KUKA KRL program: MyProgram_147().src

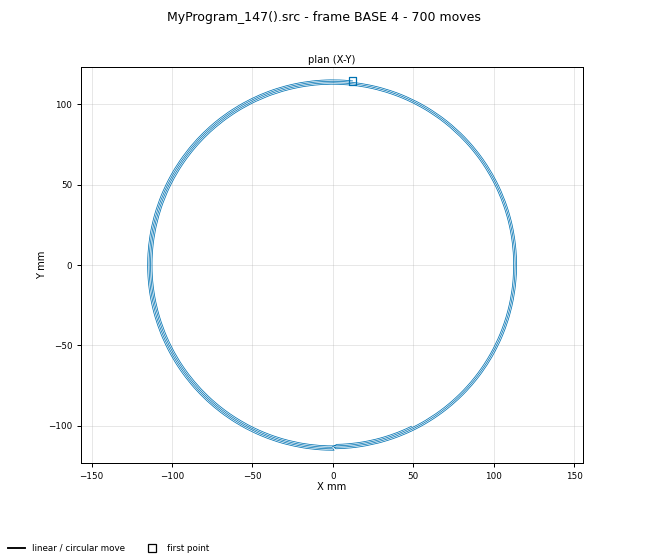
[picture p0: tool path of MyProgram_147().src in frame BASE 4, 700 of 700 moves have a stored position in this frame; points joined in program order, loops and branches not executed]
&ACCESS RVP
&REL 1
&PARAM TEMPLATE = C:\KRC\Roboter\Template\vorgabe
&PARAM EDITMASK = *
DEF MyProgram_147()
; ---- Setting reference (Base) ----
$BASE = BASE_DATA[4]

; --------------------------
; ---- Setting tool (TCP) ----
$TOOL = TOOL_DATA[3]
; --------------------------

$VEL.CP = VEL_APROX_PRINT
Startdeposition()
$VEL.CP = VEL_PRINT
LIN {X 12.2329,Y 114.5089,Z 116,A 79.5823,B 24.9341,C -1.8753,E1 25.0169,E2 366.2981} C_DIS
LIN {X 9.8806,Y 114.7378,Z 116,A 80.9993,B 24.9333,C -1.8859,E1 25.0129,E2 364.8568} C_DIS
LIN {X 7.0618,Y 114.9457,Z 116,A 82.4053,B 24.9333,C -1.8859,E1 25.0089,E2 363.4514} C_DIS
LIN {X 4.2388,Y 115.0844,Z 116,A 83.812,B 24.9333,C -1.8859,E1 25.005,E2 362.0453} C_DIS
LIN {X 1.3378,Y 115.1542,Z 116,A 85.1896,B 24.9335,C -1.8828,E1 25.0012,E2 360.6752} C_DIS
LIN {X -1.4132,Y 115.1537,Z 116,A 86.6253,B 24.9334,C -1.8854,E1 24.9972,E2 359.2332} C_DIS
LIN {X -4.2388,Y 115.0844,Z 116,A 88.0326,B 24.9334,C -1.885,E1 24.9932,E2 357.8267} C_DIS
LIN {X -7.0618,Y 114.9457,Z 116,A 89.4367,B 24.9334,C -1.8844,E1 24.9893,E2 356.4236} C_DIS
LIN {X -9.9557,Y 114.7308,Z 116,A 90.8528,B 24.9336,C -1.8826,E1 24.9854,E2 355.0113} C_DIS
LIN {X -12.7684,Y 114.452,Z 116,A 92.2606,B 24.9336,C -1.8819,E1 24.9815,E2 353.6042} C_DIS
LIN {X -15.5836,Y 114.1027,Z 116,A 93.7775,B 24.9334,C -1.8856,E1 24.9773,E2 352.0775} C_DIS
LIN {X -18.2945,Y 113.7,Z 116,A 95.072,B 24.9336,C -1.8816,E1 24.9737,E2 350.7912} C_DIS
LIN {X -21.0793,Y 113.2168,Z 116,A 96.4806,B 24.9336,C -1.8807,E1 24.9698,E2 349.3834} C_DIS
LIN {X -23.8514,Y 112.6654,Z 116,A 97.8569,B 24.9339,C -1.8782,E1 24.9661,E2 348.0114} C_DIS
LIN {X -26.6092,Y 112.0461,Z 116,A 99.2985,B 24.9339,C -1.8784,E1 24.9622,E2 346.5674} C_DIS
LIN {X -29.4238,Y 111.3397,Z 116,A 100.7129,B 24.934,C -1.8757,E1 24.9583,E2 345.1574} C_DIS
LIN {X -32.6132,Y 110.4458,Z 116,A 102.1625,B 24.9348,C -1.8656,E1 24.9545,E2 343.7295} C_DIS
LIN {X -34.8515,Y 109.7618,Z 116,A 103.4978,B 24.9343,C -1.8714,E1 24.9509,E2 342.378} C_DIS
LIN {X -37.5347,Y 108.8734,Z 116,A 104.9418,B 24.9343,C -1.8713,E1 24.9471,E2 340.9315} C_DIS
LIN {X -40.1953,Y 107.9195,Z 116,A 106.3522,B 24.9345,C -1.8696,E1 24.9434,E2 339.5222} C_DIS
LIN {X -42.8317,Y 106.9006,Z 116,A 107.7627,B 24.9345,C -1.8679,E1 24.9397,E2 338.1129} C_DIS
LIN {X -45.3731,Y 105.8474,Z 116,A 109.1681,B 24.9346,C -1.8674,E1 24.9361,E2 336.7052} C_DIS
LIN {X -48.0254,Y 104.6701,Z 116,A 110.5497,B 24.935,C -1.8627,E1 24.9326,E2 335.3316} C_DIS
LIN {X -50.5121,Y 103.4935,Z 116,A 111.9577,B 24.935,C -1.8621,E1 24.9291,E2 333.9213} C_DIS
LIN {X -53.1035,Y 102.1876,Z 116,A 113.4063,B 24.9352,C -1.86,E1 24.9255,E2 332.4739} C_DIS
LIN {X -55.5294,Y 100.8903,Z 116,A 114.7802,B 24.9353,C -1.8578,E1 24.9221,E2 331.1013} C_DIS
LIN {X -58.2622,Y 99.3355,Z 116,A 116.2478,B 24.9358,C -1.851,E1 24.9186,E2 329.6454} C_DIS
LIN {X -60.8906,Y 97.7458,Z 116,A 117.682,B 24.9362,C -1.8443,E1 24.9152,E2 328.2229} C_DIS
LIN {X -62.8639,Y 96.4905,Z 116,A 119.0192,B 24.9359,C -1.8492,E1 24.912,E2 326.8696} C_DIS
LIN {X -65.151,Y 94.9617,Z 116,A 120.4282,B 24.9359,C -1.8481,E1 24.9087,E2 325.4585} C_DIS
LIN {X -67.5228,Y 93.2896,Z 116,A 121.8441,B 24.9363,C -1.844,E1 24.9055,E2 324.0474} C_DIS
LIN {X -69.7321,Y 91.6505,Z 116,A 123.2858,B 24.9363,C -1.8442,E1 24.9023,E2 322.6003} C_DIS
LIN {X -71.9603,Y 89.9116,Z 116,A 124.6663,B 24.9365,C -1.84,E1 24.8993,E2 321.2244} C_DIS
LIN {X -74.1452,Y 88.1185,Z 116,A 126.0793,B 24.9367,C -1.8372,E1 24.8963,E2 319.8128} C_DIS
LIN {X -76.2854,Y 86.2724,Z 116,A 127.5247,B 24.9368,C -1.8356,E1 24.8932,E2 318.3655} C_DIS
LIN {X -78.4346,Y 84.3226,Z 116,A 128.9092,B 24.9372,C -1.8298,E1 24.8904,E2 316.9893} C_DIS
LIN {X -80.4267,Y 82.4253,Z 116,A 130.3516,B 24.9372,C -1.8295,E1 24.8875,E2 315.5414} C_DIS
LIN {X -82.4776,Y 80.3724,Z 116,A 131.7363,B 24.9377,C -1.8236,E1 24.8848,E2 314.165} C_DIS
LIN {X -84.3742,Y 78.3797,Z 116,A 133.1469,B 24.9377,C -1.8218,E1 24.8821,E2 312.7524} C_DIS
LIN {X -86.322,Y 76.2286,Z 116,A 134.5984,B 24.938,C -1.8185,E1 24.8794,E2 311.3024} C_DIS
LIN {X -88.1185,Y 74.1452,Z 116,A 135.975,B 24.9382,C -1.8152,E1 24.8769,E2 309.9273} C_DIS
LIN {X -89.9584,Y 71.9011,Z 116,A 137.427,B 24.9385,C -1.8118,E1 24.8743,E2 308.4768} C_DIS
LIN {X -91.6958,Y 69.6718,Z 116,A 138.8415,B 24.9387,C -1.8083,E1 24.8719,E2 307.0638} C_DIS
LIN {X -93.3342,Y 67.4619,Z 116,A 140.218,B 24.9389,C -1.8049,E1 24.8697,E2 305.6888} C_DIS
LIN {X -95.0009,Y 65.0932,Z 116,A 141.6704,B 24.9392,C -1.8013,E1 24.8674,E2 304.2377} C_DIS
LIN {X -96.5727,Y 62.7375,Z 116,A 143.0854,B 24.9394,C -1.7976,E1 24.8652,E2 302.8245} C_DIS
LIN {X -98.0441,Y 60.413,Z 116,A 144.4953,B 24.9396,C -1.7953,E1 24.8631,E2 301.4127} C_DIS
LIN {X -99.4972,Y 57.9887,Z 116,A 145.8778,B 24.9399,C -1.7903,E1 24.8611,E2 300.0351} C_DIS
LIN {X -100.8903,Y 55.5294,Z 116,A 147.4168,B 24.9399,C -1.7916,E1 24.859,E2 298.4851} C_DIS
LIN {X -102.257,Y 52.9696,Z 116,A 148.7117,B 24.9405,C -1.7813,E1 24.8574,E2 297.2078} C_DIS
LIN {X -103.5262,Y 50.4441,Z 116,A 150.1271,B 24.9408,C -1.7774,E1 24.8556,E2 295.794} C_DIS
LIN {X -104.733,Y 47.8883,Z 116,A 151.5769,B 24.941,C -1.7749,E1 24.8539,E2 294.3422} C_DIS
LIN {X -105.8474,Y 45.3731,Z 116,A 152.9548,B 24.9412,C -1.7711,E1 24.8524,E2 292.9658} C_DIS
LIN {X -106.929,Y 42.7618,Z 116,A 154.4259,B 24.9413,C -1.7694,E1 24.8508,E2 291.4906} C_DIS
LIN {X -107.9462,Y 40.1247,Z 116,A 155.8183,B 24.9417,C -1.7644,E1 24.8495,E2 290.1021} C_DIS
LIN {X -108.9055,Y 37.4426,Z 116,A 157.236,B 24.9419,C -1.76,E1 24.8482,E2 288.6869} C_DIS
LIN {X -109.785,Y 34.7797,Z 116,A 158.6502,B 24.9422,C -1.7564,E1 24.847,E2 287.2732} C_DIS
LIN {X -110.6055,Y 32.075,Z 116,A 160.066,B 24.9425,C -1.7523,E1 24.8458,E2 285.859} C_DIS
LIN {X -111.3781,Y 29.2779,Z 116,A 161.487,B 24.9428,C -1.7468,E1 24.8448,E2 284.4428} C_DIS
LIN {X -112.1254,Y 26.2662,Z 116,A 162.9247,B 24.9434,C -1.7376,E1 24.8439,E2 283.0187} C_DIS
LIN {X -112.6654,Y 23.8514,Z 116,A 164.3141,B 24.9433,C -1.74,E1 24.843,E2 281.6154} C_DIS
LIN {X -113.2168,Y 21.0793,Z 116,A 165.7301,B 24.9435,C -1.7358,E1 24.8423,E2 280.2009} C_DIS
LIN {X -113.7,Y 18.2945,Z 116,A 167.1465,B 24.9438,C -1.7317,E1 24.8417,E2 278.786} C_DIS
LIN {X -114.1812,Y 14.9855,Z 116,A 168.604,B 24.9447,C -1.718,E1 24.8411,E2 277.3523} C_DIS
LIN {X -114.4686,Y 12.6184,Z 116,A 169.9837,B 24.9444,C -1.7219,E1 24.8406,E2 275.9551} C_DIS
LIN {X -114.7378,Y 9.8806,Z 116,A 171.3948,B 24.9446,C -1.7192,E1 24.8403,E2 274.5421} C_DIS
LIN {X -114.9457,Y 7.0618,Z 116,A 172.8108,B 24.9449,C -1.715,E1 24.84,E2 273.1276} C_DIS
LIN {X -115.0844,Y 4.2388,Z 116,A 174.2271,B 24.9451,C -1.7108,E1 24.8399,E2 271.7126} C_DIS
LIN {X -115.1548,Y 1.2669,Z 116,A 175.6689,B 24.9456,C -1.7045,E1 24.8398,E2 270.2772} C_DIS
LIN {X -115.1537,Y -1.4132,Z 116,A 177.0592,B 24.9456,C -1.7025,E1 24.8398,E2 268.8834} C_DIS
LIN {X -115.0844,Y -4.2388,Z 116,A 178.6075,B 24.9456,C -1.7037,E1 24.84,E2 267.3229} C_DIS
LIN {X -114.9457,Y -7.0618,Z 116,A 179.8914,B 24.9462,C -1.6942,E1 24.8402,E2 266.054} C_DIS
LIN {X -114.7378,Y -9.8806,Z 116,A -178.7251,B 24.9466,C -1.6887,E1 24.8405,E2 264.6751} C_DIS
LIN {X -114.4607,Y -12.6935,Z 116,A -177.2766,B 24.9467,C -1.6859,E1 24.8409,E2 263.2246} C_DIS
LIN {X -114.1147,Y -15.4986,Z 116,A -175.8606,B 24.947,C -1.6818,E1 24.8414,E2 261.8099} C_DIS
LIN {X -113.7,Y -18.2945,Z 116,A -174.3898,B 24.9471,C -1.68,E1 24.842,E2 260.3348} C_DIS
LIN {X -113.2168,Y -21.0793,Z 116,A -173.0286,B 24.9475,C -1.6737,E1 24.8427,E2 258.9805} C_DIS
LIN {X -112.6654,Y -23.8514,Z 116,A -171.6455,B 24.9478,C -1.6684,E1 24.8435,E2 257.602} C_DIS
LIN {X -112.0461,Y -26.6092,Z 116,A -170.1971,B 24.948,C -1.6657,E1 24.8444,E2 256.1515} C_DIS
LIN {X -111.3397,Y -29.4238,Z 116,A -168.7763,B 24.9483,C -1.6603,E1 24.8454,E2 254.7352} C_DIS
LIN {X -110.584,Y -32.1473,Z 116,A -167.3609,B 24.9486,C -1.6564,E1 24.8465,E2 253.3209} C_DIS
LIN {X -109.7618,Y -34.8515,Z 116,A -165.9798,B 24.9489,C -1.6511,E1 24.8476,E2 251.9445} C_DIS
LIN {X -108.8984,Y -37.4635,Z 116,A -164.5353,B 24.9489,C -1.6501,E1 24.8489,E2 250.4943} C_DIS
LIN {X -107.8663,Y -40.3358,Z 116,A -163.142,B 24.9496,C -1.6405,E1 24.8502,E2 249.116} C_DIS
LIN {X -106.929,Y -42.7618,Z 116,A -161.6443,B 24.9493,C -1.6449,E1 24.8518,E2 247.5992} C_DIS
LIN {X -105.8474,Y -45.3731,Z 116,A -160.2896,B 24.9497,C -1.6387,E1 24.8533,E2 246.2517} C_DIS
LIN {X -104.6701,Y -48.0254,Z 116,A -158.9038,B 24.9501,C -1.6322,E1 24.8548,E2 244.8739} C_DIS
LIN {X -103.4935,Y -50.5121,Z 116,A -157.4923,B 24.9502,C -1.6301,E1 24.8566,E2 243.4598} C_DIS
LIN {X -102.2227,Y -53.0367,Z 116,A -156.0453,B 24.9503,C -1.6279,E1 24.8584,E2 242.0104} C_DIS
LIN {X -100.8903,Y -55.5294,Z 116,A -154.663,B 24.9506,C -1.623,E1 24.8602,E2 240.6324} C_DIS
LIN {X -99.2144,Y -58.4671,Z 116,A -153.1707,B 24.9514,C -1.6107,E1 24.8623,E2 239.1617} C_DIS
LIN {X -98.0441,Y -60.413,Z 116,A -151.8018,B 24.951,C -1.6175,E1 24.8643,E2 237.7696} C_DIS
LIN {X -96.4905,Y -62.8639,Z 116,A -150.4166,B 24.9514,C -1.6113,E1 24.8664,E2 236.3922} C_DIS
LIN {X -94.9186,Y -65.213,Z 116,A -149.0024,B 24.9516,C -1.608,E1 24.8686,E2 234.9787} C_DIS
LIN {X -93.2896,Y -67.5228,Z 116,A -147.5543,B 24.9516,C -1.6062,E1 24.871,E2 233.5278} C_DIS
LIN {X -91.6045,Y -69.7919,Z 116,A -146.1748,B 24.9519,C -1.6016,E1 24.8733,E2 232.1526} C_DIS
LIN {X -89.6717,Y -72.2564,Z 116,A -144.7035,B 24.9524,C -1.5943,E1 24.8758,E2 230.6918} C_DIS
LIN {X -88.0413,Y -74.2358,Z 116,A -143.3457,B 24.9524,C -1.5947,E1 24.8782,E2 229.3268} C_DIS
LIN {X -86.2724,Y -76.2854,Z 116,A -141.9056,B 24.9524,C -1.5954,E1 24.8809,E2 227.8785} C_DIS
LIN {X -84.3226,Y -78.4346,Z 116,A -140.5216,B 24.9526,C -1.5897,E1 24.8835,E2 226.502} C_DIS
LIN {X -82.4253,Y -80.4267,Z 116,A -139.0797,B 24.9526,C -1.5897,E1 24.8863,E2 225.0537} C_DIS
LIN {X -80.3724,Y -82.4776,Z 116,A -137.6961,B 24.953,C -1.5842,E1 24.889,E2 223.6776} C_DIS
LIN {X -78.3797,Y -84.3742,Z 116,A -136.1188,B 24.9526,C -1.5901,E1 24.8923,E2 222.0797} C_DIS
LIN {X -76.1041,Y -86.4307,Z 116,A -134.8247,B 24.9534,C -1.5774,E1 24.8949,E2 220.8108} C_DIS
LIN {X -74.1452,Y -88.1185,Z 116,A -133.4626,B 24.9534,C -1.578,E1 24.8979,E2 219.4418} C_DIS
LIN {X -71.9011,Y -89.9584,Z 116,A -131.8975,B 24.9532,C -1.5805,E1 24.9013,E2 217.8651} C_DIS
LIN {X -69.7321,Y -91.6505,Z 116,A -130.4675,B 24.9532,C -1.5805,E1 24.9045,E2 216.4296} C_DIS
LIN {X -67.4005,Y -93.378,Z 116,A -129.2239,B 24.9538,C -1.5696,E1 24.9072,E2 215.2078} C_DIS
LIN {X -65.0886,Y -95.004,Z 116,A -127.6193,B 24.9535,C -1.5757,E1 24.911,E2 213.5832} C_DIS
LIN {X -62.8009,Y -96.532,Z 116,A -126.3729,B 24.9539,C -1.5683,E1 24.9138,E2 212.3503} C_DIS
LIN {X -60.413,Y -98.0441,Z 116,A -124.994,B 24.9541,C -1.565,E1 24.9171,E2 210.975} C_DIS
LIN {X -57.9233,Y -99.5348,Z 116,A -123.4021,B 24.9539,C -1.5692,E1 24.921,E2 209.3683} C_DIS
LIN {X -55.5294,Y -100.8903,Z 116,A -122.1408,B 24.9542,C -1.5627,E1 24.924,E2 208.1187} C_DIS
LIN {X -52.9696,Y -102.257,Z 116,A -120.7254,B 24.9544,C -1.5596,E1 24.9275,E2 206.7067} C_DIS
LIN {X -50.4441,Y -103.5262,Z 116,A -119.3494,B 24.9546,C -1.5566,E1 24.9309,E2 205.3343} C_DIS
LIN {X -47.957,Y -104.702,Z 116,A -117.9108,B 24.9546,C -1.558,E1 24.9346,E2 203.8888} C_DIS
LIN {X -45.3036,Y -105.8767,Z 116,A -116.496,B 24.9546,C -1.5552,E1 24.9382,E2 202.4773} C_DIS
LIN {X -42.6916,Y -106.9566,Z 116,A -115.1207,B 24.9548,C -1.5524,E1 24.9418,E2 201.1055} C_DIS
LIN {X -40.1247,Y -107.9462,Z 116,A -113.683,B 24.9548,C -1.5541,E1 24.9455,E2 199.6609} C_DIS
LIN {X -37.392,Y -108.9225,Z 116,A -112.3028,B 24.955,C -1.5502,E1 24.9491,E2 198.2874} C_DIS
LIN {X -34.7797,Y -109.785,Z 116,A -110.898,B 24.955,C -1.5506,E1 24.9529,E2 196.8788} C_DIS
LIN {X -32.075,Y -110.6055,Z 116,A -109.4894,B 24.955,C -1.5498,E1 24.9567,E2 195.47} C_DIS
LIN {X -29.3509,Y -111.3593,Z 116,A -108.0489,B 24.955,C -1.5504,E1 24.9606,E2 194.0258} C_DIS
LIN {X -26.5357,Y -112.0631,Z 116,A -106.6356,B 24.955,C -1.5483,E1 24.9644,E2 192.6156} C_DIS
LIN {X -23.8213,Y -112.6716,Z 116,A -105.2312,B 24.955,C -1.5485,E1 24.9682,E2 191.2089} C_DIS
LIN {X -21.0694,Y -113.2186,Z 116,A -103.8253,B 24.955,C -1.5485,E1 24.9721,E2 189.8017} C_DIS
LIN {X -18.2945,Y -113.7,Z 116,A -102.4186,B 24.955,C -1.5482,E1 24.976,E2 188.3941} C_DIS
LIN {X -15.405,Y -114.1269,Z 116,A -101.0051,B 24.9552,C -1.5462,E1 24.9799,E2 186.9844} C_DIS
LIN {X -12.6184,Y -114.4686,Z 116,A -99.6,B 24.9552,C -1.5463,E1 24.9838,E2 185.5779} C_DIS
LIN {X -9.8806,Y -114.7378,Z 116,A -98.1986,B 24.9552,C -1.5477,E1 24.9877,E2 184.1727} C_DIS
LIN {X -7.0618,Y -114.9457,Z 116,A -96.7926,B 24.9552,C -1.5477,E1 24.9916,E2 182.7661} C_DIS
LIN {X -4.2388,Y -115.0844,Z 116,A -95.3864,B 24.9552,C -1.5478,E1 24.9955,E2 181.3593} C_DIS
LIN {X -1.3378,Y -115.1542,Z 116,A -93.9828,B 24.9552,C -1.5463,E1 24.9994,E2 179.9593} C_DIS
LIN {X 0.8075,Y -115.1575,Z 116,A -93.2725,B 24.9561,C -1.5308,E1 25.0013,E2 179.2858} C_DIS
Enddeposition()
LIN {X 0.8075,Y -115.1575,Z 116,A -93.2725,B 24.9561,C -1.5308,E1 25.0013,E2 179.2858} C_DIS
Startdeposition()
$VEL.CP = VEL_PRINT
LIN {X 0.0523,Y -114.2549,Z 116,A -93.9442,B 24.9559,C -1.5337,E1 24.9995,E2 179.9505} C_DIS
LIN {X -2.8973,Y -114.218,Z 116,A -95.3914,B 24.9559,C -1.5349,E1 24.9954,E2 181.395} C_DIS
LIN {X -5.7835,Y -114.1077,Z 116,A -96.9837,B 24.9562,C -1.5285,E1 24.9909,E2 183.0027} C_DIS
LIN {X -8.4348,Y -113.9433,Z 116,A -98.3985,B 24.9564,C -1.5249,E1 24.987,E2 184.4267} C_DIS
LIN {X -12.3662,Y -113.5829,Z 116,A -100.3944,B 24.9564,C -1.5244,E1 24.9814,E2 186.4248} C_DIS
LIN {X -16.6336,Y -113.0372,Z 116,A -102.6291,B 24.9566,C -1.5216,E1 24.9752,E2 188.6681} C_DIS
LIN {X -20.6313,Y -112.3757,Z 116,A -104.5197,B 24.9562,C -1.5283,E1 24.97,E2 190.5445} C_DIS
LIN {X -26.3827,Y -111.1669,Z 116,A -107.816,B 24.957,C -1.5149,E1 24.961,E2 193.8768} C_DIS
LIN {X -29.6836,Y -110.3298,Z 116,A -109.0853,B 24.9559,C -1.5345,E1 24.9577,E2 195.1015} C_DIS
LIN {X -32.779,Y -109.4504,Z 116,A -110.6791,B 24.9558,C -1.5365,E1 24.9534,E2 196.6932} C_DIS
LIN {X -35.2511,Y -108.6791,Z 116,A -112.0991,B 24.956,C -1.5323,E1 24.9496,E2 198.1256} C_DIS
LIN {X -38.4354,Y -107.596,Z 116,A -113.8668,B 24.9561,C -1.5303,E1 24.9449,E2 199.9015} C_DIS
LIN {X -42.4746,Y -106.0665,Z 116,A -115.7998,B 24.9554,C -1.5422,E1 24.9399,E2 201.8103} C_DIS
LIN {X -44.5782,Y -105.1979,Z 116,A -116.9365,B 24.9554,C -1.5436,E1 24.937,E2 202.9463} C_DIS
LIN {X -47.2556,Y -104.0231,Z 116,A -118.5876,B 24.9557,C -1.5375,E1 24.9327,E2 204.616} C_DIS
LIN {X -54.6973,Y -100.3097,Z 116,A -122.1859,B 24.954,C -1.5667,E1 24.9239,E2 208.1544} C_DIS
LIN {X -58.7436,Y -97.9971,Z 116,A -125.1729,B 24.9554,C -1.5429,E1 24.9165,E2 211.207} C_DIS
LIN {X -62.0172,Y -95.9571,Z 116,A -126.9361,B 24.9548,C -1.553,E1 24.9124,E2 212.9518} C_DIS
LIN {X -65.2993,Y -93.7539,Z 116,A -129.0411,B 24.9549,C -1.5512,E1 24.9075,E2 215.0681} C_DIS
LIN {X -68.1158,Y -91.7301,Z 116,A -130.6101,B 24.9543,C -1.5612,E1 24.904,E2 216.6188} C_DIS
LIN {X -71.0705,Y -89.4586,Z 116,A -132.6896,B 24.9546,C -1.556,E1 24.8994,E2 218.7185} C_DIS
LIN {X -73.7987,Y -87.222,Z 116,A -134.3858,B 24.9543,C -1.5623,E1 24.8958,E2 220.406} C_DIS
LIN {X -76.325,Y -85.0194,Z 116,A -136.0658,B 24.9541,C -1.5657,E1 24.8923,E2 222.0846} C_DIS
LIN {X -78.6689,Y -82.8569,Z 116,A -138.1645,B 24.9551,C -1.5487,E1 24.8879,E2 224.2325} C_DIS
LIN {X -81.4176,Y -80.156,Z 116,A -139.5391,B 24.9535,C -1.5755,E1 24.8853,E2 225.5491} C_DIS
LIN {X -83.4797,Y -78.0067,Z 116,A -141.6839,B 24.9548,C -1.5524,E1 24.8811,E2 227.7582} C_DIS
LIN {X -86.3351,Y -74.8345,Z 116,A -143.1469,B 24.9529,C -1.5847,E1 24.8786,E2 229.151} C_DIS
LIN {X -88.0105,Y -72.8558,Z 116,A -144.5946,B 24.9531,C -1.5817,E1 24.8759,E2 230.6123} C_DIS
LIN {X -90.008,Y -70.3753,Z 116,A -146.3137,B 24.9531,C -1.5806,E1 24.8729,E2 232.3422} C_DIS
LIN {X -92.033,Y -67.7035,Z 116,A -147.6863,B 24.9522,C -1.5973,E1 24.8707,E2 233.6818} C_DIS
LIN {X -93.4091,Y -65.7951,Z 116,A -148.9697,B 24.9522,C -1.596,E1 24.8686,E2 234.9744} C_DIS
LIN {X -95.3134,Y -63.0011,Z 116,A -150.6397,B 24.9519,C -1.6014,E1 24.866,E2 236.6398} C_DIS
LIN {X -97.0339,Y -60.318,Z 116,A -152.3243,B 24.9519,C -1.6022,E1 24.8635,E2 238.3312} C_DIS
LIN {X -99.0863,Y -56.8831,Z 116,A -154.3917,B 24.9517,C -1.6051,E1 24.8605,E2 240.4022} C_DIS
LIN {X -100.8693,Y -53.6599,Z 116,A -156.3422,B 24.9517,C -1.6061,E1 24.8579,E2 242.3608} C_DIS
LIN {X -102.6639,Y -50.1432,Z 116,A -158.357,B 24.9514,C -1.6102,E1 24.8554,E2 244.3766} C_DIS
LIN {X -104.1486,Y -46.977,Z 116,A -159.9468,B 24.9507,C -1.6218,E1 24.8536,E2 245.9475} C_DIS
LIN {X -105.5075,Y -43.8436,Z 116,A -161.6412,B 24.9504,C -1.6275,E1 24.8517,E2 247.6377} C_DIS
LIN {X -106.6002,Y -41.1176,Z 116,A -163.6601,B 24.9514,C -1.6102,E1 24.8497,E2 249.7092} C_DIS
LIN {X -107.8471,Y -37.72,Z 116,A -164.5942,B 24.9489,C -1.6506,E1 24.8489,E2 250.5523} C_DIS
LIN {X -108.5086,Y -35.7778,Z 116,A -166.1285,B 24.95,C -1.6335,E1 24.8475,E2 252.1361} C_DIS
LIN {X -109.6395,Y -32.1418,Z 116,A -168.3669,B 24.9504,C -1.6264,E1 24.8456,E2 254.4044} C_DIS
LIN {X -110.553,Y -28.8441,Z 116,A -169.7762,B 24.9494,C -1.6437,E1 24.8447,E2 255.7804} C_DIS
LIN {X -111.5051,Y -24.9142,Z 116,A -171.6192,B 24.9485,C -1.6573,E1 24.8435,E2 257.6018} C_DIS
LIN {X -111.9864,Y -22.6478,Z 116,A -172.8536,B 24.9485,C -1.6581,E1 24.8428,E2 258.8416} C_DIS
LIN {X -112.6514,Y -19.0653,Z 116,A -174.6711,B 24.9481,C -1.6643,E1 24.8419,E2 260.6552} C_DIS
LIN {X -113.1208,Y -16.0456,Z 116,A -176.3353,B 24.9481,C -1.664,E1 24.8412,E2 262.3302} C_DIS
LIN {X -113.5477,Y -12.6906,Z 116,A -177.9551,B 24.9476,C -1.6724,E1 24.8407,E2 263.9396} C_DIS
LIN {X -113.8898,Y -9.1044,Z 116,A -179.7787,B 24.9473,C -1.6775,E1 24.8402,E2 265.7618} C_DIS
LIN {X -114.0942,Y -6.0299,Z 116,A 178.5178,B 24.9473,C -1.6763,E1 24.8399,E2 267.4785} C_DIS
LIN {X -114.2279,Y -2.4208,Z 116,A 176.8972,B 24.9465,C -1.6896,E1 24.8399,E2 269.077} C_DIS
LIN {X -114.2486,Y 1.0733,Z 116,A 175.1131,B 24.9462,C -1.6941,E1 24.8399,E2 270.8614} C_DIS
LIN {X -114.1847,Y 3.9815,Z 116,A 173.617,B 24.946,C -1.6973,E1 24.8399,E2 272.3587} C_DIS
LIN {X -114.0016,Y 7.5781,Z 116,A 171.7908,B 24.9457,C -1.7024,E1 24.8402,E2 274.1837} C_DIS
LIN {X -113.7057,Y 11.1926,Z 116,A 169.9812,B 24.9453,C -1.7087,E1 24.8407,E2 275.9893} C_DIS
LIN {X -113.3931,Y 14.0084,Z 116,A 168.3462,B 24.9455,C -1.7049,E1 24.8412,E2 277.6432} C_DIS
LIN {X -112.8959,Y 17.5581,Z 116,A 166.5235,B 24.9452,C -1.7097,E1 24.842,E2 279.4651} C_DIS
LIN {X -112.1731,Y 21.7017,Z 116,A 164.6057,B 24.9443,C -1.7241,E1 24.8429,E2 281.36} C_DIS
LIN {X -111.5102,Y 24.8908,Z 116,A 162.9848,B 24.9439,C -1.7298,E1 24.8438,E2 282.9768} C_DIS
LIN {X -110.7383,Y 28.1232,Z 116,A 161.236,B 24.9438,C -1.7319,E1 24.845,E2 284.7308} C_DIS
LIN {X -110.084,Y 30.5879,Z 116,A 159.8245,B 24.9438,C -1.7307,E1 24.8461,E2 286.1533} C_DIS
LIN {X -108.7107,Y 35.1534,Z 116,A 157.595,B 24.943,C -1.7447,E1 24.8479,E2 288.3624} C_DIS
LIN {X -107.7954,Y 37.8671,Z 116,A 156.1407,B 24.9427,C -1.7485,E1 24.8492,E2 289.816} C_DIS
LIN {X -106.7199,Y 40.8016,Z 116,A 154.5429,B 24.9425,C -1.7521,E1 24.8508,E2 291.4141} C_DIS
LIN {X -104.5438,Y 46.0933,Z 116,A 151.6842,B 24.9419,C -1.7613,E1 24.8539,E2 294.2666} C_DIS
LIN {X -103.4573,Y 48.4814,Z 116,A 150.4001,B 24.9415,C -1.7666,E1 24.8553,E2 295.5452} C_DIS
LIN {X -102.395,Y 50.6856,Z 116,A 149.1304,B 24.9414,C -1.7686,E1 24.8569,E2 296.817} C_DIS
LIN {X -99.725,Y 55.7558,Z 116,A 146.5818,B 24.9399,C -1.79,E1 24.8602,E2 299.3282} C_DIS
LIN {X -97.5652,Y 59.4543,Z 116,A 143.5713,B 24.9418,C -1.7621,E1 24.8646,E2 302.4208} C_DIS
LIN {X -95.6264,Y 62.5264,Z 116,A 142.1036,B 24.9405,C -1.7812,E1 24.8668,E2 303.8504} C_DIS
LIN {X -93.4169,Y 65.784,Z 116,A 140.0523,B 24.9404,C -1.7836,E1 24.87,E2 305.9061} C_DIS
LIN {X -90.9507,Y 69.1533,Z 116,A 138.1517,B 24.9395,C -1.7969,E1 24.8732,E2 307.7839} C_DIS
LIN {X -89.575,Y 70.9232,Z 116,A 136.9861,B 24.9394,C -1.7983,E1 24.8752,E2 308.9518} C_DIS
LIN {X -87.8799,Y 73.0129,Z 116,A 135.5179,B 24.9394,C -1.7972,E1 24.8778,E2 310.4296} C_DIS
LIN {X -85.7024,Y 75.5589,Z 116,A 133.9808,B 24.9388,C -1.8072,E1 24.8806,E2 311.9497} C_DIS
LIN {X -84.0682,Y 77.3715,Z 116,A 132.5685,B 24.9391,C -1.8028,E1 24.8833,E2 313.3788} C_DIS
LIN {X -81.7346,Y 79.8351,Z 116,A 131.0549,B 24.9383,C -1.8145,E1 24.8862,E2 314.8711} C_DIS
LIN {X -79.3629,Y 82.1907,Z 116,A 129.2055,B 24.9385,C -1.8116,E1 24.8899,E2 316.735} C_DIS
LIN {X -76.8963,Y 84.5042,Z 116,A 127.5354,B 24.9381,C -1.8166,E1 24.8933,E2 318.4} C_DIS
LIN {X -74.2104,Y 86.8712,Z 116,A 125.9058,B 24.9374,C -1.8274,E1 24.8967,E2 320.0104} C_DIS
LIN {X -72.3878,Y 88.3967,Z 116,A 124.4479,B 24.938,C -1.8193,E1 24.8999,E2 321.493} C_DIS
LIN {X -69.7922,Y 90.459,Z 116,A 122.8423,B 24.9376,C -1.8252,E1 24.9034,E2 323.0905} C_DIS
LIN {X -66.2263,Y 93.1014,Z 116,A 120.5704,B 24.9374,C -1.8279,E1 24.9085,E2 325.3638} C_DIS
LIN {X -63.5442,Y 94.9541,Z 116,A 119.0965,B 24.9367,C -1.8377,E1 24.9119,E2 326.8195} C_DIS
LIN {X -61.6596,Y 96.1866,Z 116,A 117.8077,B 24.937,C -1.8334,E1 24.9149,E2 328.1227} C_DIS
LIN {X -58.533,Y 98.1217,Z 116,A 115.8952,B 24.937,C -1.834,E1 24.9195,E2 330.0396} C_DIS
LIN {X -55.1532,Y 100.0614,Z 116,A 114.1583,B 24.9361,C -1.8463,E1 24.9237,E2 331.7524} C_DIS
LIN {X -52.6623,Y 101.3947,Z 116,A 112.2413,B 24.9373,C -1.8283,E1 24.9286,E2 333.7174} C_DIS
LIN {X -49.6432,Y 102.9046,Z 116,A 111.2538,B 24.9352,C -1.8598,E1 24.9309,E2 334.6325} C_DIS
LIN {X -46.8367,Y 104.2118,Z 116,A 109.2498,B 24.9363,C -1.8437,E1 24.936,E2 336.6798} C_DIS
LIN {X -43.705,Y 105.5652,Z 116,A 107.5473,B 24.9361,C -1.8465,E1 24.9404,E2 338.3796} C_DIS
LIN {X -39.7633,Y 107.1125,Z 116,A 105.4064,B 24.9359,C -1.8486,E1 24.946,E2 340.52} C_DIS
LIN {X -35.73,Y 108.5241,Z 116,A 103.5205,B 24.935,C -1.8618,E1 24.9509,E2 342.378} C_DIS
LIN {X -32.5626,Y 109.5146,Z 116,A 101.7356,B 24.9352,C -1.8588,E1 24.9557,E2 344.1733} C_DIS
LIN {X -29.336,Y 110.4237,Z 116,A 100.1019,B 24.935,C -1.8625,E1 24.9601,E2 345.8007} C_DIS
LIN {X -26.1215,Y 111.2277,Z 116,A 98.3223,B 24.9352,C -1.8592,E1 24.9649,E2 347.5906} C_DIS
LIN {X -22.8852,Y 111.9377,Z 116,A 96.6499,B 24.9352,C -1.8602,E1 24.9695,E2 349.2626} C_DIS
LIN {X -19.5103,Y 112.577,Z 116,A 95.07,B 24.9346,C -1.8674,E1 24.9738,E2 350.827} C_DIS
LIN {X -16.6306,Y 113.0377,Z 116,A 92.6975,B 24.9372,C -1.8306,E1 24.9806,E2 353.2888} C_DIS
LIN {X -11.3395,Y 113.6904,Z 116,A 90.7969,B 24.9349,C -1.8642,E1 24.9857,E2 355.1108} C_DIS
LIN {X -8.0871,Y 113.9672,Z 116,A 89.1646,B 24.9348,C -1.8651,E1 24.9902,E2 356.7417} C_DIS
LIN {X -4.6028,Y 114.1607,Z 116,A 87.4382,B 24.9347,C -1.8667,E1 24.995,E2 358.4647} C_DIS
LIN {X -1.0742,Y 114.2487,Z 116,A 85.3087,B 24.9357,C -1.852,E1 25.0011,E2 360.6291} C_DIS
LIN {X 2.2581,Y 114.2309,Z 116,A 83.75,B 24.9354,C -1.857,E1 25.0054,E2 362.1758} C_DIS
LIN {X 7.177,Y 114.0287,Z 116,A 81.5079,B 24.9347,C -1.8666,E1 25.0116,E2 364.3942} C_DIS
LIN {X 11.7811,Y 113.6441,Z 116,A 79.2353,B 24.9346,C -1.8683,E1 25.0179,E2 366.6616} C_DIS
LIN {X 17.1976,Y 112.9517,Z 116,A 76.7614,B 24.9338,C -1.879,E1 25.0247,E2 369.108} C_DIS
LIN {X 22.8155,Y 111.952,Z 116,A 73.7294,B 24.9344,C -1.8705,E1 25.033,E2 372.1568} C_DIS
LIN {X 27.1126,Y 110.9895,Z 116,A 71.4537,B 24.9347,C -1.8664,E1 25.0392,E2 374.439} C_DIS
LIN {X 30.0103,Y 110.2416,Z 116,A 69.9895,B 24.9347,C -1.867,E1 25.0432,E2 375.8995} C_DIS
LIN {X 33.482,Y 109.2376,Z 116,A 68.2904,B 24.9344,C -1.8706,E1 25.0477,E2 377.5872} C_DIS
LIN {X 35.6356,Y 108.5546,Z 116,A 66.8511,B 24.9354,C -1.8564,E1 25.0516,E2 379.0575} C_DIS
LIN {X 39.7797,Y 107.1065,Z 116,A 64.8635,B 24.9349,C -1.8637,E1 25.0568,E2 381.0238} C_DIS
LIN {X 42.4794,Y 106.0645,Z 116,A 63.1691,B 24.9357,C -1.8516,E1 25.0612,E2 382.743} C_DIS
LIN {X 45.6215,Y 104.7495,Z 116,A 60.3551,B 24.9391,C -1.8018,E1 25.0688,E2 385.6678} C_DIS
LIN {X 52.2755,Y 101.593,Z 116,A 58.1911,B 24.9349,C -1.8637,E1 25.0738,E2 387.6796} C_DIS
LIN {X 54.5297,Y 100.4006,Z 116,A 56.6592,B 24.9358,C -1.8508,E1 25.0776,E2 389.2378} C_DIS
LIN {X 58.1915,Y 98.3235,Z 116,A 54.4154,B 24.9364,C -1.8419,E1 25.083,E2 391.4958} C_DIS
LIN {X 61.3574,Y 96.3806,Z 116,A 51.6173,B 24.9394,C -1.7979,E1 25.0899,E2 394.3888} C_DIS
LIN {X 66.7975,Y 92.6939,Z 116,A 49.5384,B 24.9361,C -1.8458,E1 25.0943,E2 396.3473} C_DIS
LIN {X 68.6691,Y 91.3145,Z 116,A 48.3285,B 24.9364,C -1.8418,E1 25.097,E2 397.5623} C_DIS
LIN {X 71.5294,Y 89.0932,Z 116,A 46.5038,B 24.9367,C -1.838,E1 25.101,E2 399.3891} C_DIS
LIN {X 74.0272,Y 87.0273,Z 116,A 44.7504,B 24.9373,C -1.8292,E1 25.1048,E2 401.1567} C_DIS
LIN {X 79.3077,Y 82.2439,Z 116,A 41.2884,B 24.9374,C -1.8268,E1 25.1119,E2 404.6102} C_DIS
LIN {X 81.9425,Y 79.6204,Z 116,A 39.3686,B 24.9379,C -1.8203,E1 25.1157,E2 406.5373} C_DIS
LIN {X 84.6661,Y 76.7195,Z 116,A 37.5183,B 24.9378,C -1.8223,E1 25.1192,E2 408.3747} C_DIS
LIN {X 87.2436,Y 73.7733,Z 116,A 34.5569,B 24.9411,C -1.7729,E1 25.1247,E2 411.4392} C_DIS
LIN {X 90.9285,Y 69.1828,Z 116,A 32.6244,B 24.9385,C -1.8115,E1 25.1279,E2 413.2715} C_DIS
LIN {X 93.1704,Y 66.1297,Z 116,A 30.5598,B 24.9393,C -1.7993,E1 25.1313,E2 415.355} C_DIS
LIN {X 95.7964,Y 62.2675,Z 116,A 28.4282,B 24.9391,C -1.8028,E1 25.1345,E2 417.4677} C_DIS
LIN {X 99.2992,Y 56.5125,Z 116,A 25.0793,B 24.9396,C -1.795,E1 25.1394,E2 420.8177} C_DIS
LIN {X 100.5212,Y 54.3075,Z 116,A 23.7336,B 24.9401,C -1.7878,E1 25.1412,E2 422.1734} C_DIS
LIN {X 101.8676,Y 51.7382,Z 116,A 22.366,B 24.9401,C -1.7878,E1 25.1429,E2 423.5339} C_DIS
LIN {X 103.0649,Y 49.3096,Z 116,A 20.6863,B 24.9413,C -1.7692,E1 25.145,E2 425.2485} C_DIS
LIN {X 104.6048,Y 45.9533,Z 116,A 17.9028,B 24.9445,C -1.7215,E1 25.1483,E2 428.1291} C_DIS
LIN {X 107.2,Y 39.5232,Z 116,A 15.6339,B 24.9415,C -1.7662,E1 25.1504,E2 430.2801} C_DIS
LIN {X 108.09,Y 37.0219,Z 116,A 14.4445,B 24.9414,C -1.7687,E1 25.1514,E2 431.4568} C_DIS
LIN {X 109.1009,Y 33.9229,Z 116,A 12.8193,B 24.9417,C -1.7642,E1 25.1528,E2 433.0835} C_DIS
LIN {X 109.9776,Y 30.9635,Z 116,A 11.2229,B 24.9421,C -1.7572,E1 25.1541,E2 434.6872} C_DIS
LIN {X 110.8414,Y 27.72,Z 116,A 9.5602,B 24.9424,C -1.7529,E1 25.1552,E2 436.3505} C_DIS
LIN {X 111.4644,Y 25.0972,Z 116,A 8.089,B 24.9431,C -1.7432,E1 25.1562,E2 437.8361} C_DIS
LIN {X 112.2014,Y 21.5552,Z 116,A 6.3116,B 24.9433,C -1.7392,E1 25.1571,E2 439.6125} C_DIS
LIN {X 113.0772,Y 16.3512,Z 116,A 3.5539,B 24.9442,C -1.7256,E1 25.1584,E2 442.3859} C_DIS
LIN {X 113.5905,Y 12.2934,Z 116,A 1.286,B 24.9453,C -1.709,E1 25.1591,E2 444.6796} C_DIS
LIN {X 113.8993,Y 8.9848,Z 116,A 0.0175,B 24.9444,C -1.7221,E1 25.1594,E2 445.9098} C_DIS
LIN {X 114.1268,Y 5.3928,Z 116,A -1.8509,B 24.945,C -1.7133,E1 25.1597,E2 447.7879} C_DIS
LIN {X 114.242,Y 1.6558,Z 116,A -3.6962,B 24.9453,C -1.7085,E1 25.1597,E2 449.6333} C_DIS
LIN {X 114.228,Y -2.4167,Z 116,A -5.5717,B 24.9453,C -1.7096,E1 25.1597,E2 451.4951} C_DIS
LIN {X 114.1183,Y -5.5828,Z 116,A -7.2702,B 24.9459,C -1.6993,E1 25.1595,E2 453.2078} C_DIS
LIN {X 113.8937,Y -9.0547,Z 116,A -9.0163,B 24.9462,C -1.6936,E1 25.1592,E2 454.957} C_DIS
LIN {X 113.5876,Y -12.3208,Z 116,A -10.647,B 24.9465,C -1.6889,E1 25.1587,E2 456.5891} C_DIS
LIN {X 113.2406,Y -15.1853,Z 116,A -13.0431,B 24.9496,C -1.6404,E1 25.1578,E2 459.0853} C_DIS
LIN {X 112.2766,Y -21.1645,Z 116,A -14.933,B 24.9469,C -1.6835,E1 25.1569,E2 460.8627} C_DIS
LIN {X 111.2646,Y -25.9621,Z 116,A -17.4553,B 24.9476,C -1.6726,E1 25.1554,E2 463.396} C_DIS
LIN {X 110.4085,Y -29.3923,Z 116,A -19.0804,B 24.9476,C -1.6738,E1 25.1543,E2 465.009} C_DIS
LIN {X 109.7885,Y -31.6307,Z 116,A -20.3477,B 24.948,C -1.6653,E1 25.1533,E2 466.2891} C_DIS
LIN {X 109.1136,Y -33.8821,Z 116,A -21.493,B 24.9482,C -1.6631,E1 25.1524,E2 467.433} C_DIS
LIN {X 108.0894,Y -37.0237,Z 116,A -23.1744,B 24.9486,C -1.6567,E1 25.1509,E2 469.1199} C_DIS
LIN {X 107.2326,Y -39.434,Z 116,A -24.6381,B 24.9493,C -1.6443,E1 25.1495,E2 470.6047} C_DIS
LIN {X 106.0178,Y -42.5941,Z 116,A -26.0596,B 24.9489,C -1.6518,E1 25.1481,E2 472.0005} C_DIS
LIN {X 104.9331,Y -45.2002,Z 116,A -27.4575,B 24.9491,C -1.6483,E1 25.1466,E2 473.3991} C_DIS
LIN {X 103.5994,Y -48.1761,Z 116,A -30.2264,B 24.9526,C -1.5912,E1 25.1432,E2 476.2878} C_DIS
LIN {X 100.8852,Y -53.6297,Z 116,A -32.4573,B 24.9508,C -1.6197,E1 25.1404,E2 478.4395} C_DIS
LIN {X 98.8767,Y -57.2478,Z 116,A -34.2379,B 24.9504,C -1.6273,E1 25.138,E2 480.1931} C_DIS
LIN {X 97.2996,Y -59.8913,Z 116,A -35.8045,B 24.9507,C -1.6217,E1 25.1357,E2 481.7648} C_DIS
LIN {X 95.9576,Y -62.0165,Z 116,A -37.0697,B 24.951,C -1.6179,E1 25.1338,E2 483.0326} C_DIS
LIN {X 94.3525,Y -64.4328,Z 116,A -38.5119,B 24.9512,C -1.6143,E1 25.1315,E2 484.476} C_DIS
LIN {X 92.8234,Y -66.6159,Z 116,A -39.8161,B 24.9513,C -1.6121,E1 25.1294,E2 485.7791} C_DIS
LIN {X 91.1968,Y -68.8258,Z 116,A -41.357,B 24.952,C -1.6008,E1 25.1268,E2 487.3395} C_DIS
LIN {X 89.0432,Y -71.591,Z 116,A -43.0275,B 24.952,C -1.6,E1 25.1239,E2 489.0039} C_DIS
LIN {X 86.6008,Y -74.5278,Z 116,A -44.8453,B 24.952,C -1.5995,E1 25.1207,E2 490.8147} C_DIS
LIN {X 84.7751,Y -76.5979,Z 116,A -46.2035,B 24.9522,C -1.5971,E1 25.1182,E2 492.1724} C_DIS
LIN {X 83.2058,Y -78.2979,Z 116,A -47.3927,B 24.9525,C -1.5928,E1 25.1159,E2 493.3665} C_DIS
LIN {X 80.9821,Y -80.5969,Z 116,A -49.1535,B 24.9531,C -1.5816,E1 25.1124,E2 495.1461} C_DIS
LIN {X 77.8662,Y -83.6118,Z 116,A -51.4487,B 24.9538,C -1.5709,E1 25.1077,E2 497.4572} C_DIS
LIN {X 74.0679,Y -86.9926,Z 116,A -53.704,B 24.9533,C -1.5785,E1 25.103,E2 499.6858} C_DIS
LIN {X 71.406,Y -89.1932,Z 116,A -55.5206,B 24.9538,C -1.5707,E1 25.0991,E2 501.5139} C_DIS
LIN {X 68.6503,Y -91.3285,Z 116,A -57.2259,B 24.9538,C -1.5689,E1 25.0953,E2 503.2171} C_DIS
LIN {X 66.1038,Y -93.1888,Z 116,A -58.7669,B 24.954,C -1.5674,E1 25.0918,E2 504.7562} C_DIS
LIN {X 62.9167,Y -95.3691,Z 116,A -60.7568,B 24.9543,C -1.5611,E1 25.0872,E2 506.7543} C_DIS
LIN {X 60.3062,Y -97.0412,Z 116,A -62.1705,B 24.9541,C -1.5645,E1 25.0839,E2 508.1555} C_DIS
LIN {X 57.363,Y -98.8105,Z 116,A -63.8212,B 24.9541,C -1.5645,E1 25.0799,E2 509.8011} C_DIS
LIN {X 54.3319,Y -100.5079,Z 116,A -65.8086,B 24.955,C -1.5504,E1 25.075,E2 511.8162} C_DIS
LIN {X 51.3666,Y -102.0574,Z 116,A -67.313,B 24.9547,C -1.5553,E1 25.0713,E2 513.3048} C_DIS
LIN {X 48.829,Y -103.2953,Z 116,A -68.9624,B 24.9554,C -1.5425,E1 25.0671,E2 514.9801} C_DIS
LIN {X 45.5647,Y -104.7742,Z 116,A -71.3439,B 24.9571,C -1.5139,E1 25.0608,E2 517.4236} C_DIS
LIN {X 40.8691,Y -106.6943,Z 116,A -73.6325,B 24.9566,C -1.5216,E1 25.0549,E2 519.6888} C_DIS
LIN {X 37.1088,Y -108.0607,Z 116,A -75.2477,B 24.9558,C -1.5363,E1 25.0507,E2 521.266} C_DIS
LIN {X 33.7691,Y -109.1486,Z 116,A -76.9358,B 24.9558,C -1.5375,E1 25.0463,E2 522.9483} C_DIS
LIN {X 30.5774,Y -110.087,Z 116,A -78.4699,B 24.9555,C -1.5416,E1 25.0422,E2 524.4701} C_DIS
LIN {X 28.0199,Y -110.7648,Z 116,A -79.9198,B 24.9559,C -1.5348,E1 25.0382,E2 525.934} C_DIS
LIN {X 20.8866,Y -112.3293,Z 116,A -83.9185,B 24.9569,C -1.5167,E1 25.0272,E2 529.9705} C_DIS
LIN {X 17.5985,Y -112.8897,Z 116,A -85.5667,B 24.9569,C -1.5166,E1 25.0226,E2 531.6173} C_DIS
LIN {X 14.2426,Y -113.3628,Z 116,A -86.7951,B 24.9558,C -1.5361,E1 25.0194,E2 532.7986} C_DIS
LIN {X 11.3793,Y -113.6862,Z 116,A -89.1704,B 24.9581,C -1.4948,E1 25.0125,E2 535.2702} C_DIS
LIN {X 6.0602,Y -114.0925,Z 116,A -91.2524,B 24.9568,C -1.5193,E1 25.0069,E2 537.2932} C_DIS
LIN {X 1.8746,Y -114.2379,Z 116,A -93.0886,B 24.9561,C -1.5301,E1 25.0018,E2 539.1035} C_DIS
LIN {X 1.8746,Y -114.2379,Z 116,A -93.0886,B 24.9561,C -1.5301,E1 25.0018,E2 539.1035} C_DIS
Enddeposition()
LIN {X 0.7978,Y -113.3424,Z 116,A -93.5858,B 24.9551,C -1.5478,E1 25.0006,E2 539.5587} C_DIS
Startdeposition()
$VEL.CP = VEL_PRINT
LIN {X 7.942,Y -113.0678,Z 116,A -89.3215,B 24.9534,C -1.5773,E1 25.0126,E2 535.2255} C_DIS
LIN {X 13.6506,Y -112.5219,Z 116,A -86.4623,B 24.9534,C -1.5772,E1 25.0206,E2 532.3686} C_DIS
LIN {X 20.6494,Y -111.4507,Z 116,A -82.6916,B 24.9527,C -1.5883,E1 25.031,E2 528.5754} C_DIS
LIN {X 25.2707,Y -110.4933,Z 116,A -80.637,B 24.9535,C -1.5758,E1 25.0365,E2 526.5531} C_DIS
LIN {X 28.1593,Y -109.7924,Z 116,A -78.927,B 24.9528,C -1.5865,E1 25.0412,E2 524.8201} C_DIS
LIN {X 31.7553,Y -108.8079,Z 116,A -76.9691,B 24.9525,C -1.5919,E1 25.0465,E2 522.8529} C_DIS
LIN {X 35.0001,Y -107.8068,Z 116,A -75.3702,B 24.9527,C -1.5887,E1 25.0507,E2 521.2644} C_DIS
LIN {X 38.7486,Y -106.5169,Z 116,A -73.0635,B 24.9517,C -1.6049,E1 25.0569,E2 518.924} C_DIS
LIN {X 44.0397,Y -104.4404,Z 116,A -70.494,B 24.9523,C -1.5953,E1 25.0635,E2 516.3831} C_DIS
LIN {X 47.0394,Y -103.1255,Z 116,A -68.7978,B 24.9521,C -1.5997,E1 25.0678,E2 514.6808} C_DIS
LIN {X 49.717,Y -101.8627,Z 116,A -67.414,B 24.9522,C -1.597,E1 25.0713,E2 513.3069} C_DIS
LIN {X 52.1962,Y -100.6148,Z 116,A -65.8981,B 24.9518,C -1.6045,E1 25.0751,E2 511.7775} C_DIS
LIN {X 55.2051,Y -98.9934,Z 116,A -64.2493,B 24.9518,C -1.604,E1 25.0791,E2 510.1347} C_DIS
LIN {X 58.0632,Y -97.3456,Z 116,A -62.5747,B 24.9516,C -1.6074,E1 25.0831,E2 508.4572} C_DIS
LIN {X 62.5572,Y -94.5195,Z 116,A -60.3684,B 24.9526,C -1.5909,E1 25.0883,E2 506.2968} C_DIS
LIN {X 64.5725,Y -93.1543,Z 116,A -58.6057,B 24.951,C -1.6176,E1 25.0924,E2 504.4771} C_DIS
LIN {X 67.9751,Y -90.7012,Z 116,A -56.5054,B 24.9508,C -1.6211,E1 25.0972,E2 502.376} C_DIS
LIN {X 70.8728,Y -88.4576,Z 116,A -54.6486,B 24.9505,C -1.6254,E1 25.1012,E2 500.5161} C_DIS
LIN {X 73.4898,Y -86.2934,Z 116,A -53.0256,B 24.9505,C -1.625,E1 25.1047,E2 498.9002} C_DIS
LIN {X 76.1079,Y -83.9955,Z 116,A -51.3484,B 24.9505,C -1.6253,E1 25.1082,E2 497.229} C_DIS
LIN {X 78.4037,Y -81.8553,Z 116,A -49.65,B 24.95,C -1.6342,E1 25.1117,E2 495.5165} C_DIS
LIN {X 80.7395,Y -79.5516,Z 116,A -48.0594,B 24.9499,C -1.6352,E1 25.1148,E2 493.9303} C_DIS
LIN {X 83.3114,Y -76.8544,Z 116,A -46.131,B 24.9495,C -1.642,E1 25.1185,E2 491.9942} C_DIS
LIN {X 85.5299,Y -74.3774,Z 116,A -44.5254,B 24.9495,C -1.6429,E1 25.1214,E2 490.3938} C_DIS
LIN {X 87.5871,Y -71.946,Z 116,A -42.7741,B 24.9488,C -1.6537,E1 25.1246,E2 488.6251} C_DIS
LIN {X 89.8223,Y -69.1322,Z 116,A -41.1202,B 24.9489,C -1.6511,E1 25.1274,E2 486.9852} C_DIS
LIN {X 91.9675,Y -66.2536,Z 116,A -39.1694,B 24.9482,C -1.6624,E1 25.1307,E2 485.0171} C_DIS
LIN {X 94.2455,Y -62.9728,Z 116,A -36.8071,B 24.9469,C -1.684,E1 25.1344,E2 482.6153} C_DIS
LIN {X 96.1672,Y -59.9932,Z 116,A -35.5122,B 24.948,C -1.666,E1 25.1363,E2 481.3695} C_DIS
LIN {X 97.794,Y -57.3046,Z 116,A -33.8092,B 24.9474,C -1.676,E1 25.1387,E2 479.6517} C_DIS
LIN {X 100.8799,Y -51.6775,Z 116,A -30.6588,B 24.947,C -1.6812,E1 25.1429,E2 476.5054} C_DIS
LIN {X 103.4129,Y -46.4015,Z 116,A -27.6799,B 24.9464,C -1.6912,E1 25.1464,E2 473.5192} C_DIS
LIN {X 105.0037,Y -42.6794,Z 116,A -25.7378,B 24.9464,C -1.6926,E1 25.1485,E2 471.5843} C_DIS
LIN {X 106.2485,Y -39.4839,Z 116,A -24.0678,B 24.9462,C -1.695,E1 25.1502,E2 469.9179} C_DIS
LIN {X 107.1659,Y -36.9215,Z 116,A -22.6958,B 24.9459,C -1.6992,E1 25.1514,E2 468.5438} C_DIS
LIN {X 108.0069,Y -34.3816,Z 116,A -21.2167,B 24.9452,C -1.7094,E1 25.1527,E2 467.049} C_DIS
LIN {X 108.9834,Y -31.1446,Z 116,A -19.3246,B 24.9443,C -1.7234,E1 25.1542,E2 465.1347} C_DIS
LIN {X 109.8845,Y -27.8008,Z 116,A -17.8002,B 24.9447,C -1.7184,E1 25.1553,E2 463.6309} C_DIS
LIN {X 110.8958,Y -23.4444,Z 116,A -15.4407,B 24.9439,C -1.7303,E1 25.1567,E2 461.257} C_DIS
LIN {X 112.1449,Y -16.4653,Z 116,A -11.9877,B 24.9435,C -1.7358,E1 25.1583,E2 457.8115} C_DIS
LIN {X 112.5999,Y -12.9847,Z 116,A -9.7613,B 24.9418,C -1.7628,E1 25.159,E2 455.5345} C_DIS
LIN {X 112.9807,Y -9.0919,Z 116,A -7.9702,B 24.9419,C -1.7605,E1 25.1594,E2 453.7595} C_DIS
LIN {X 113.193,Y -5.8972,Z 116,A -6.8983,B 24.9432,C -1.7402,E1 25.1596,E2 452.7419} C_DIS
LIN {X 113.3415,Y 1.0605,Z 116,A -2.7288,B 24.9405,C -1.7821,E1 25.1597,E2 448.4983} C_DIS
LIN {X 113.244,Y 4.8069,Z 116,A -1.3188,B 24.9416,C -1.7655,E1 25.1596,E2 447.1358} C_DIS
LIN {X 113.0612,Y 8.0383,Z 116,A 0.7568,B 24.9399,C -1.7914,E1 25.1592,E2 445.0115} C_DIS
LIN {X 112.7433,Y 11.6738,Z 116,A 2.1776,B 24.9408,C -1.7775,E1 25.1588,E2 443.632} C_DIS
LIN {X 111.8528,Y 18.3405,Z 116,A 5.5373,B 24.9402,C -1.7864,E1 25.1575,E2 440.271} C_DIS
LIN {X 111.2998,Y 21.4396,Z 116,A 7.1222,B 24.9399,C -1.7911,E1 25.1567,E2 438.6842} C_DIS
LIN {X 110.4808,Y 25.3247,Z 116,A 9.1005,B 24.9395,C -1.7961,E1 25.1555,E2 436.7057} C_DIS
LIN {X 109.5894,Y 28.946,Z 116,A 11.0351,B 24.939,C -1.8042,E1 25.1541,E2 434.7632} C_DIS
LIN {X 108.5048,Y 32.7768,Z 116,A 12.9077,B 24.939,C -1.8039,E1 25.1527,E2 432.902} C_DIS
LIN {X 107.5493,Y 35.7862,Z 116,A 14.5329,B 24.9386,C -1.81,E1 25.1513,E2 431.2714} C_DIS
LIN {X 105.9281,Y 40.3309,Z 116,A 17.2938,B 24.9371,C -1.8322,E1 25.1486,E2 428.4736} C_DIS
LIN {X 103.8218,Y 45.4793,Z 116,A 19.7492,B 24.9376,C -1.8239,E1 25.1459,E2 426.0513} C_DIS
LIN {X 102.0971,Y 49.2291,Z 116,A 21.6678,B 24.9378,C -1.8221,E1 25.1437,E2 424.1473} C_DIS
LIN {X 100.8694,Y 51.698,Z 116,A 23.1735,B 24.9371,C -1.8312,E1 25.1418,E2 422.6282} C_DIS
LIN {X 99.3273,Y 54.6059,Z 116,A 24.9547,B 24.9365,C -1.8412,E1 25.1394,E2 420.8329} C_DIS
LIN {X 96.2467,Y 59.8659,Z 116,A 27.8707,B 24.9365,C -1.8419,E1 25.1352,E2 417.9301} C_DIS
LIN {X 94.5793,Y 62.4665,Z 116,A 29.5193,B 24.9359,C -1.8499,E1 25.1327,E2 416.2708} C_DIS
LIN {X 92.2614,Y 65.8418,Z 116,A 31.5249,B 24.9357,C -1.8523,E1 25.1295,E2 414.2695} C_DIS
LIN {X 90.2066,Y 68.6335,Z 116,A 33.6377,B 24.9342,C -1.8731,E1 25.1259,E2 412.1177} C_DIS
LIN {X 86.7491,Y 72.9544,Z 116,A 36.1278,B 24.9348,C -1.8657,E1 25.1215,E2 409.6565} C_DIS
LIN {X 84.4301,Y 75.6232,Z 116,A 38.3194,B 24.9332,C -1.8883,E1 25.1174,E2 407.4213} C_DIS
LIN {X 81.8753,Y 78.3829,Z 116,A 39.5373,B 24.935,C -1.8614,E1 25.1152,E2 406.2721} C_DIS
LIN {X 79.3477,Y 80.9409,Z 116,A 41.7851,B 24.9334,C -1.8848,E1 25.1106,E2 403.9787} C_DIS
LIN {X 74.2048,Y 85.6807,Z 116,A 44.9329,B 24.9341,C -1.8744,E1 25.1042,E2 400.868} C_DIS
LIN {X 70.8832,Y 88.4492,Z 116,A 47.3835,B 24.933,C -1.8905,E1 25.0988,E2 398.3888} C_DIS
LIN {X 68.0242,Y 90.6643,Z 116,A 49.0955,B 24.9331,C -1.8886,E1 25.0951,E2 396.6874} C_DIS
LIN {X 63.2552,Y 94.0543,Z 116,A 52.2379,B 24.9322,C -1.9018,E1 25.0878,E2 393.5246} C_DIS
LIN {X 59.4177,Y 96.5259,Z 116,A 54.5357,B 24.932,C -1.905,E1 25.0824,E2 391.2267} C_DIS
LIN {X 55.7816,Y 98.6715,Z 116,A 56.6062,B 24.932,C -1.9052,E1 25.0774,E2 389.1618} C_DIS
LIN {X 52.8019,Y 100.2959,Z 116,A 58.1196,B 24.9324,C -1.8986,E1 25.0737,E2 387.6683} C_DIS
LIN {X 47.9753,Y 102.6921,Z 116,A 60.9974,B 24.9317,C -1.9088,E1 25.0664,E2 384.7741} C_DIS
LIN {X 43.6096,Y 104.6217,Z 116,A 63.3209,B 24.9317,C -1.9075,E1 25.0605,E2 382.4593} C_DIS
LIN {X 40.8598,Y 105.7269,Z 116,A 64.7046,B 24.932,C -1.9039,E1 25.0569,E2 381.0869} C_DIS
LIN {X 38.1952,Y 106.7188,Z 116,A 66.2233,B 24.9317,C -1.9088,E1 25.0529,E2 379.5599} C_DIS
LIN {X 35.1468,Y 107.7593,Z 116,A 67.8123,B 24.9317,C -1.9085,E1 25.0487,E2 377.9747} C_DIS
LIN {X 32.2583,Y 108.6587,Z 116,A 69.5601,B 24.9309,C -1.9192,E1 25.044,E2 376.2046} C_DIS
LIN {X 28.2568,Y 109.7673,Z 116,A 71.4673,B 24.9314,C -1.9122,E1 25.0389,E2 374.317} C_DIS
LIN {X 24.3902,Y 110.6909,Z 116,A 73.3955,B 24.9316,C -1.9098,E1 25.0337,E2 372.3973} C_DIS
LIN {X 21.6933,Y 111.251,Z 116,A 74.8797,B 24.9313,C -1.9144,E1 25.0296,E2 370.9041} C_DIS
LIN {X 18.4481,Y 111.8348,Z 116,A 76.5061,B 24.9313,C -1.9132,E1 25.0251,E2 369.282} C_DIS
LIN {X 13.1737,Y 112.5778,Z 116,A 79.197,B 24.9313,C -1.9138,E1 25.0177,E2 366.5921} C_DIS
LIN {X 7.8985,Y 113.0707,Z 116,A 82.0092,B 24.9309,C -1.9197,E1 25.0098,E2 363.7673} C_DIS
LIN {X 0.2064,Y 113.3468,Z 116,A 85.9801,B 24.9307,C -1.9226,E1 24.9987,E2 359.7902} C_DIS
LIN {X -5.6099,Y 113.2089,Z 116,A 88.8739,B 24.9309,C -1.9197,E1 24.9907,E2 356.903} C_DIS
LIN {X -10.9273,Y 112.8191,Z 116,A 91.6509,B 24.9308,C -1.9219,E1 24.9829,E2 354.1194} C_DIS
LIN {X -16.1383,Y 112.1913,Z 116,A 93.9104,B 24.9321,C -1.9037,E1 24.9768,E2 351.9014} C_DIS
LIN {X -18.7842,Y 111.7786,Z 116,A 95.403,B 24.9317,C -1.9086,E1 24.9726,E2 350.3959} C_DIS
LIN {X -22.2817,Y 111.1355,Z 116,A 97.3183,B 24.9315,C -1.912,E1 24.9673,E2 348.4703} C_DIS
LIN {X -25.7072,Y 110.3924,Z 116,A 99.0085,B 24.9318,C -1.907,E1 24.9628,E2 346.7898} C_DIS
LIN {X -29.3161,Y 109.4894,Z 116,A 100.9057,B 24.9319,C -1.9058,E1 24.9576,E2 344.8927} C_DIS
LIN {X -34.372,Y 108.01,Z 116,A 103.5848,B 24.9321,C -1.9035,E1 24.9505,E2 342.2146} C_DIS
LIN {X -37.9943,Y 106.7894,Z 116,A 105.6261,B 24.9319,C -1.9056,E1 24.9451,E2 340.1644} C_DIS
LIN {X -41.3091,Y 105.5504,Z 116,A 107.2322,B 24.9326,C -1.8957,E1 24.9409,E2 338.5785} C_DIS
LIN {X -46.3002,Y 103.4586,Z 116,A 110.0779,B 24.9326,C -1.8962,E1 24.9336,E2 335.7249} C_DIS
LIN {X -49.6583,Y 101.8909,Z 116,A 112.2032,B 24.9321,C -1.9036,E1 24.9282,E2 333.5766} C_DIS
LIN {X -56.9426,Y 98.0058,Z 116,A 116.0281,B 24.9336,C -1.882,E1 24.9189,E2 329.7921} C_DIS
LIN {X -61.7718,Y 95.0362,Z 116,A 119.1061,B 24.9334,C -1.8852,E1 24.9116,E2 326.6967} C_DIS
LIN {X -64.2009,Y 93.4126,Z 116,A 120.499,B 24.9338,C -1.8789,E1 24.9084,E2 325.3143} C_DIS
LIN {X -66.8573,Y 91.5282,Z 116,A 122.1154,B 24.9341,C -1.8743,E1 24.9048,E2 323.7031} C_DIS
LIN {X -69.4565,Y 89.5724,Z 116,A 123.9655,B 24.9338,C -1.8791,E1 24.9006,E2 321.8348} C_DIS
LIN {X -72.8217,Y 86.8594,Z 116,A 126.028,B 24.9345,C -1.8693,E1 24.8962,E2 319.7879} C_DIS
LIN {X -75.6394,Y 84.4156,Z 116,A 127.886,B 24.9349,C -1.8639,E1 24.8923,E2 317.9355} C_DIS
LIN {X -78.7383,Y 81.5328,Z 116,A 130.1907,B 24.9348,C -1.8655,E1 24.8876,E2 315.6174} C_DIS
LIN {X -81.9185,Y 78.3381,Z 116,A 132.3711,B 24.9354,C -1.8559,E1 24.8834,E2 313.4506} C_DIS
LIN {X -84.4203,Y 75.6341,Z 116,A 134.205,B 24.9358,C -1.85,E1 24.88,E2 311.6224} C_DIS
LIN {X -86.7862,Y 72.9096,Z 116,A 136.1794,B 24.9358,C -1.8513,E1 24.8764,E2 309.6359} C_DIS
LIN {X -90.1236,Y 68.7412,Z 116,A 138.6795,B 24.9368,C -1.8361,E1 24.8721,E2 307.1603} C_DIS
LIN {X -91.6593,Y 66.6784,Z 116,A 140.0077,B 24.937,C -1.8337,E1 24.8699,E2 305.8314} C_DIS
LIN {X -93.4408,Y 64.1602,Z 116,A 142.1244,B 24.9357,C -1.8517,E1 24.8665,E2 303.6614} C_DIS
LIN {X -95.5398,Y 60.9879,Z 116,A 143.7949,B 24.9368,C -1.8361,E1 24.864,E2 302.0196} C_DIS
LIN {X -98.6423,Y 55.834,Z 116,A 146.523,B 24.9383,C -1.8148,E1 24.8602,E2 299.3282} C_DIS
LIN {X -100.1798,Y 53.0221,Z 116,A 148.3294,B 24.9381,C -1.8174,E1 24.8578,E2 297.5059} C_DIS
LIN {X -102.1199,Y 49.1818,Z 116,A 150.4807,B 24.9386,C -1.8099,E1 24.8551,E2 295.3608} C_DIS
LIN {X -103.8009,Y 45.5273,Z 116,A 153.1132,B 24.9374,C -1.8277,E1 24.8521,E2 292.6716} C_DIS
LIN {X -105.5007,Y 41.4355,Z 116,A 155.4157,B 24.9377,C -1.8232,E1 24.8497,E2 290.3667} C_DIS
LIN {X -107.1341,Y 37.012,Z 116,A 158.0152,B 24.9377,C -1.8244,E1 24.8474,E2 287.7496} C_DIS
LIN {X -108.8044,Y 31.7671,Z 116,A 159.9436,B 24.9405,C -1.7815,E1 24.8459,E2 285.9125} C_DIS
LIN {X -110.0829,Y 27.0013,Z 116,A 162.4283,B 24.9411,C -1.7731,E1 24.8441,E2 283.4333} C_DIS
LIN {X -110.7999,Y 23.8904,Z 116,A 164.0268,B 24.9415,C -1.7674,E1 24.8432,E2 281.8391} C_DIS
LIN {X -111.4395,Y 20.7115,Z 116,A 166.1953,B 24.9404,C -1.7831,E1 24.842,E2 279.6204} C_DIS
LIN {X -112.0452,Y 17.1236,Z 116,A 167.4687,B 24.9423,C -1.7547,E1 24.8415,E2 278.4071} C_DIS
LIN {X -112.4178,Y 14.4761,Z 116,A 168.9159,B 24.9423,C -1.7541,E1 24.841,E2 276.9527} C_DIS
LIN {X -112.838,Y 10.7227,Z 116,A 170.8434,B 24.9427,C -1.7486,E1 24.8404,E2 275.0267} C_DIS
LIN {X -113.1096,Y 7.3224,Z 116,A 172.5609,B 24.9431,C -1.7427,E1 24.8401,E2 273.3129} C_DIS
LIN {X -113.285,Y 3.7243,Z 116,A 174.4408,B 24.9433,C -1.7391,E1 24.8398,E2 271.4303} C_DIS
LIN {X -113.3446,Y 0.4559,Z 116,A 176.1753,B 24.9435,C -1.737,E1 24.8398,E2 269.6903} C_DIS
LIN {X -113.2924,Y -3.4838,Z 116,A 178.0476,B 24.9442,C -1.7258,E1 24.8398,E2 267.8335} C_DIS
LIN {X -113.1323,Y -6.9878,Z 116,A -179.9801,B 24.944,C -1.7279,E1 24.8402,E2 265.8442} C_DIS
LIN {X -112.8069,Y -11.0599,Z 116,A -177.9002,B 24.9444,C -1.7219,E1 24.8407,E2 263.7662} C_DIS
LIN {X -112.3909,Y -14.6833,Z 116,A -176.2361,B 24.9453,C -1.7089,E1 24.8413,E2 262.1232} C_DIS
LIN {X -111.9933,Y -17.4592,Z 116,A -174.8072,B 24.9455,C -1.7049,E1 24.8419,E2 260.6954} C_DIS
LIN {X -111.5151,Y -20.2912,Z 116,A -173.3468,B 24.9458,C -1.7006,E1 24.8426,E2 259.2364} C_DIS
LIN {X -110.9484,Y -23.1931,Z 116,A -171.75,B 24.9458,C -1.7,E1 24.8435,E2 257.6318} C_DIS
LIN {X -110.0162,Y -27.2749,Z 116,A -169.7263,B 24.9465,C -1.6897,E1 24.8448,E2 255.6207} C_DIS
LIN {X -108.1585,Y -33.8993,Z 116,A -166.2135,B 24.9471,C -1.6804,E1 24.8475,E2 252.1098} C_DIS
LIN {X -105.9098,Y -40.3792,Z 116,A -162.7431,B 24.9477,C -1.6701,E1 24.8507,E2 248.6442} C_DIS
LIN {X -104.8499,Y -43.0573,Z 116,A -161.0937,B 24.9475,C -1.6736,E1 24.8525,E2 246.9773} C_DIS
LIN {X -103.3524,Y -46.5359,Z 116,A -159.2894,B 24.9481,C -1.6636,E1 24.8545,E2 245.1868} C_DIS
LIN {X -101.8624,Y -49.7176,Z 116,A -157.4463,B 24.9483,C -1.6613,E1 24.8567,E2 243.3393} C_DIS
LIN {X -99.5047,Y -54.2789,Z 116,A -155.0163,B 24.9491,C -1.6474,E1 24.8598,E2 240.9293} C_DIS
LIN {X -97.4473,Y -57.8912,Z 116,A -152.8434,B 24.9493,C -1.6446,E1 24.8629,E2 238.7518} C_DIS
LIN {X -95.794,Y -60.5905,Z 116,A -151.0266,B 24.949,C -1.6491,E1 24.8656,E2 236.915} C_DIS
LIN {X -93.6622,Y -63.8343,Z 116,A -149.2086,B 24.9497,C -1.6383,E1 24.8684,E2 235.1139} C_DIS
LIN {X -91.6394,Y -66.7054,Z 116,A -147.3602,B 24.9498,C -1.6368,E1 24.8714,E2 233.2599} C_DIS
LIN {X -89.463,Y -69.5985,Z 116,A -145.3093,B 24.9495,C -1.6413,E1 24.8749,E2 231.1886} C_DIS
LIN {X -86.8928,Y -72.7814,Z 116,A -143.364,B 24.9501,C -1.6314,E1 24.8784,E2 229.2579} C_DIS
LIN {X -83.0293,Y -77.1606,Z 116,A -140.4521,B 24.9506,C -1.623,E1 24.8838,E2 226.3528} C_DIS
LIN {X -80.4195,Y -79.8756,Z 116,A -138.3172,B 24.9503,C -1.6284,E1 24.888,E2 224.1959} C_DIS
LIN {X -77.6021,Y -82.6149,Z 116,A -136.6364,B 24.9513,C -1.6117,E1 24.8913,E2 222.548} C_DIS
LIN {X -75.3279,Y -84.6944,Z 116,A -135.0125,B 24.9513,C -1.6113,E1 24.8947,E2 220.9186} C_DIS
LIN {X -72.4729,Y -87.1492,Z 116,A -133.0935,B 24.9515,C -1.6083,E1 24.8988,E2 218.9993} C_DIS
LIN {X -69.3322,Y -89.6682,Z 116,A -131.069,B 24.9518,C -1.6041,E1 24.9032,E2 216.9773} C_DIS
LIN {X -66.7307,Y -91.621,Z 116,A -129.5012,B 24.9521,C -1.5981,E1 24.9067,E2 215.4183} C_DIS
LIN {X -63.9721,Y -93.5689,Z 116,A -127.6221,B 24.9519,C -1.6024,E1 24.9111,E2 213.5226} C_DIS
LIN {X -60.5675,Y -95.8084,Z 116,A -125.7588,B 24.9526,C -1.5909,E1 24.9154,E2 211.6804} C_DIS
LIN {X -58.3148,Y -97.1962,Z 116,A -124.1314,B 24.952,C -1.6011,E1 24.9194,E2 210.024} C_DIS
LIN {X -55.3068,Y -98.9367,Z 116,A -122.563,B 24.9526,C -1.5907,E1 24.9231,E2 208.4756} C_DIS
LIN {X -50.9993,Y -101.2253,Z 116,A -119.8929,B 24.9523,C -1.5961,E1 24.9298,E2 205.7854} C_DIS
LIN {X -47.4855,Y -102.9203,Z 116,A -117.9868,B 24.9526,C -1.591,E1 24.9346,E2 203.8865} C_DIS
LIN {X -43.3582,Y -104.7274,Z 116,A -115.7542,B 24.9528,C -1.5867,E1 24.9403,E2 201.6592} C_DIS
LIN {X -40.198,Y -105.9784,Z 116,A -114.1245,B 24.9531,C -1.5813,E1 24.9445,E2 200.0387} C_DIS
LIN {X -37.222,Y -107.0604,Z 116,A -112.3899,B 24.9529,C -1.5856,E1 24.9491,E2 198.2905} C_DIS
LIN {X -32.9513,Y -108.4524,Z 116,A -110.2966,B 24.9534,C -1.5763,E1 24.9547,E2 196.2156} C_DIS
LIN {X -28.9952,Y -109.5761,Z 116,A -107.9835,B 24.9529,C -1.585,E1 24.961,E2 193.8782} C_DIS
LIN {X -24.8587,Y -110.5873,Z 116,A -105.7261,B 24.9527,C -1.5884,E1 24.9671,E2 191.6097} C_DIS
LIN {X -19.4855,Y -111.66,Z 116,A -102.5364,B 24.9517,C -1.6056,E1 24.976,E2 188.3759} C_DIS
LIN {X -14.971,Y -112.3536,Z 116,A -100.3003,B 24.9519,C -1.602,E1 24.9822,E2 186.1467} C_DIS
LIN {X -10.7316,Y -112.8372,Z 116,A -98.9796,B 24.9541,C -1.5654,E1 24.9856,E2 184.9121} C_DIS
LIN {X -8.1652,Y -113.0527,Z 116,A -96.9702,B 24.9523,C -1.5961,E1 24.9914,E2 182.8289} C_DIS
LIN {X -4.487,Y -113.2577,Z 116,A -95.0625,B 24.9521,C -1.5984,E1 24.9968,E2 180.9156} C_DIS
LIN {X -0.6045,Y -113.3444,Z 116,A -93.6493,B 24.9535,C -1.5746,E1 25.0005,E2 179.5587} C_DIS
LIN {X -0.6045,Y -113.3444,Z 116,A -93.6493,B 24.9535,C -1.5746,E1 25.0005,E2 179.5587} C_DIS
Enddeposition()
LIN {X 0.8058,Y -112.4294,Z 116,A -94.1472,B 24.9556,C -1.5388,E1 24.9989,E2 180.1414} C_DIS
Startdeposition()
$VEL.CP = VEL_PRINT
LIN {X -3.1701,Y -112.3944,Z 116,A -95.9044,B 24.955,C -1.5497,E1 24.9941,E2 181.8728} C_DIS
LIN {X -8.4148,Y -112.1248,Z 116,A -98.3827,B 24.9545,C -1.558,E1 24.9872,E2 184.3323} C_DIS
LIN {X -13.8979,Y -111.5779,Z 116,A -101.0829,B 24.9542,C -1.5629,E1 24.9798,E2 187.0226} C_DIS
LIN {X -18.3257,Y -110.9356,Z 116,A -103.2092,B 24.9538,C -1.5699,E1 24.9739,E2 189.1339} C_DIS
LIN {X -20.7299,Y -110.5127,Z 116,A -104.8176,B 24.9547,C -1.555,E1 24.9694,E2 190.7795} C_DIS
LIN {X -27.2935,Y -109.0779,Z 116,A -108.0902,B 24.9542,C -1.563,E1 24.9605,E2 194.0373} C_DIS
LIN {X -31.346,Y -107.9831,Z 116,A -110.2448,B 24.9542,C -1.5637,E1 24.9547,E2 196.1935} C_DIS
LIN {X -35.8906,Y -106.5568,Z 116,A -112.7402,B 24.9542,C -1.5628,E1 24.9481,E2 198.6957} C_DIS
LIN {X -39.344,Y -105.3318,Z 116,A -114.6357,B 24.9542,C -1.5632,E1 24.9431,E2 200.5939} C_DIS
LIN {X -42.8913,Y -103.938,Z 116,A -116.5066,B 24.9539,C -1.5681,E1 24.9383,E2 202.4573} C_DIS
LIN {X -45.9115,Y -102.6388,Z 116,A -118.287,B 24.9541,C -1.5656,E1 24.9337,E2 204.2479} C_DIS
LIN {X -49.0527,Y -101.1754,Z 116,A -120.6299,B 24.9553,C -1.5442,E1 24.9277,E2 206.6476} C_DIS
LIN {X -52.99,Y -99.1716,Z 116,A -122.1902,B 24.9535,C -1.5752,E1 24.924,E2 208.1385} C_DIS
LIN {X -57.5142,Y -96.6164,Z 116,A -124.8656,B 24.9534,C -1.5779,E1 24.9175,E2 210.8155} C_DIS
LIN {X -60.6074,Y -94.7061,Z 116,A -126.8397,B 24.9534,C -1.5758,E1 24.9128,E2 212.8009} C_DIS
LIN {X -64.0261,Y -92.4293,Z 116,A -128.9492,B 24.9534,C -1.5785,E1 24.9079,E2 214.9109} C_DIS
LIN {X -66.9343,Y -90.3476,Z 116,A -130.8392,B 24.9533,C -1.5789,E1 24.9036,E2 216.8066} C_DIS
LIN {X -69.8836,Y -88.0841,Z 116,A -132.5661,B 24.9527,C -1.5892,E1 24.8999,E2 218.5155} C_DIS
LIN {X -72.7198,Y -85.7577,Z 116,A -134.4942,B 24.9527,C -1.5904,E1 24.8957,E2 220.4482} C_DIS
LIN {X -75.0214,Y -83.7512,Z 116,A -136.0355,B 24.9524,C -1.594,E1 24.8925,E2 221.9868} C_DIS
LIN {X -77.6729,Y -81.2998,Z 116,A -138.2863,B 24.9531,C -1.5814,E1 24.8878,E2 224.2768} C_DIS
LIN {X -79.9942,Y -79.0153,Z 116,A -139.1949,B 24.9511,C -1.615,E1 24.8862,E2 225.1094} C_DIS
LIN {X -81.8205,Y -77.1226,Z 116,A -141.439,B 24.9531,C -1.5819,E1 24.8817,E2 227.4419} C_DIS
LIN {X -84.4783,Y -74.2024,Z 116,A -142.6947,B 24.951,C -1.6165,E1 24.8795,E2 228.6209} C_DIS
LIN {X -85.8181,Y -72.6488,Z 116,A -143.949,B 24.9514,C -1.6106,E1 24.8772,E2 229.895} C_DIS
LIN {X -89.6911,Y -67.8093,Z 116,A -146.9338,B 24.9505,C -1.6251,E1 24.8721,E2 232.8593} C_DIS
LIN {X -92.2458,Y -64.2901,Z 116,A -149.4212,B 24.9508,C -1.6199,E1 24.868,E2 235.3713} C_DIS
LIN {X -94.3078,Y -61.228,Z 116,A -151.1803,B 24.9502,C -1.6295,E1 24.8653,E2 237.1162} C_DIS
LIN {X -95.7272,Y -58.9853,Z 116,A -152.7153,B 24.9505,C -1.6259,E1 24.863,E2 238.6677} C_DIS
LIN {X -98.2502,Y -54.6755,Z 116,A -154.9808,B 24.9494,C -1.6438,E1 24.8599,E2 240.9022} C_DIS
LIN {X -100.2996,Y -50.8196,Z 116,A -157.1544,B 24.9489,C -1.6519,E1 24.8571,E2 243.068} C_DIS
LIN {X -101.9321,Y -47.4587,Z 116,A -159.3134,B 24.9491,C -1.6473,E1 24.8544,E2 245.2498} C_DIS
LIN {X -103.3578,Y -44.2729,Z 116,A -161.0637,B 24.9488,C -1.6535,E1 24.8524,E2 246.9949} C_DIS
LIN {X -104.5425,Y -41.3937,Z 116,A -162.7528,B 24.9488,C -1.6542,E1 24.8507,E2 248.6918} C_DIS
LIN {X -106.6835,Y -35.5149,Z 116,A -166.0101,B 24.9483,C -1.661,E1 24.8476,E2 251.9513} C_DIS
LIN {X -107.9674,Y -31.3977,Z 116,A -168.487,B 24.9486,C -1.6569,E1 24.8456,E2 254.4524} C_DIS
LIN {X -108.982,Y -27.668,Z 116,A -170.4566,B 24.9482,C -1.663,E1 24.8442,E2 256.4189} C_DIS
LIN {X -110.0831,Y -22.8969,Z 116,A -172.6241,B 24.9469,C -1.6834,E1 24.843,E2 258.5504} C_DIS
LIN {X -110.6528,Y -19.9611,Z 116,A -174.1611,B 24.9466,C -1.6877,E1 24.8422,E2 260.0863} C_DIS
LIN {X -111.2282,Y -16.4685,Z 116,A -175.927,B 24.9462,C -1.6949,E1 24.8414,E2 261.8457} C_DIS
LIN {X -111.6042,Y -13.6879,Z 116,A -177.5236,B 24.9462,C -1.693,E1 24.8408,E2 263.4562} C_DIS
LIN {X -111.9643,Y -10.3187,Z 116,A -179.1727,B 24.9457,C -1.7016,E1 24.8404,E2 265.0948} C_DIS
LIN {X -112.2013,Y -7.3094,Z 116,A 179.2941,B 24.9454,C -1.7067,E1 24.8401,E2 266.625} C_DIS
LIN {X -112.3801,Y -3.6363,Z 116,A 177.2938,B 24.9454,C -1.7079,E1 24.8398,E2 268.6345} C_DIS
LIN {X -112.4364,Y 0.663,Z 116,A 175.1978,B 24.9446,C -1.7187,E1 24.8398,E2 270.7174} C_DIS
LIN {X -112.3831,Y 3.5408,Z 116,A 173.676,B 24.9445,C -1.7213,E1 24.8399,E2 272.2421} C_DIS
LIN {X -112.2315,Y 6.8549,Z 116,A 171.9511,B 24.9442,C -1.7254,E1 24.8402,E2 273.9675} C_DIS
LIN {X -111.9743,Y 10.2102,Z 116,A 170.2757,B 24.9437,C -1.7326,E1 24.8406,E2 275.636} C_DIS
LIN {X -111.6257,Y 13.5046,Z 116,A 168.586,B 24.9434,C -1.738,E1 24.8411,E2 277.3229} C_DIS
LIN {X -111.2178,Y 16.5382,Z 116,A 166.0983,B 24.9454,C -1.7076,E1 24.8422,E2 279.8979} C_DIS
LIN {X -110.2764,Y 21.9551,Z 116,A 164.2521,B 24.9424,C -1.7531,E1 24.8431,E2 281.6466} C_DIS
LIN {X -109.77,Y 24.3554,Z 116,A 162.972,B 24.9422,C -1.756,E1 24.8438,E2 282.9274} C_DIS
LIN {X -108.2292,Y 30.4787,Z 116,A 159.4654,B 24.9422,C -1.7551,E1 24.8463,E2 286.4564} C_DIS
LIN {X -106.6018,Y 35.7571,Z 116,A 157.1452,B 24.9404,C -1.7831,E1 24.8482,E2 288.7233} C_DIS
LIN {X -105.6987,Y 38.3447,Z 116,A 154.1814,B 24.9441,C -1.7275,E1 24.8512,E2 291.8363} C_DIS
LIN {X -103.1018,Y 44.8609,Z 116,A 152.1855,B 24.9394,C -1.7988,E1 24.8532,E2 293.6732} C_DIS
LIN {X -102.2361,Y 46.8051,Z 116,A 150.7131,B 24.9401,C -1.787,E1 24.8549,E2 295.1818} C_DIS
LIN {X -100.8026,Y 49.8131,Z 116,A 148.7429,B 24.9405,C -1.7817,E1 24.8573,E2 297.1754} C_DIS
LIN {X -98.4912,Y 54.2439,Z 116,A 146.4753,B 24.9393,C -1.8,E1 24.8603,E2 299.4115} C_DIS
LIN {X -95.4023,Y 59.5054,Z 116,A 143.694,B 24.9378,C -1.8217,E1 24.8642,E2 302.1553} C_DIS
LIN {X -94.1723,Y 61.4358,Z 116,A 141.7523,B 24.9396,C -1.7949,E1 24.8673,E2 304.1707} C_DIS
LIN {X -92.295,Y 64.2193,Z 116,A 140.6533,B 24.9377,C -1.8234,E1 24.8689,E2 305.2072} C_DIS
LIN {X -90.7516,Y 66.3825,Z 116,A 138.3665,B 24.9399,C -1.791,E1 24.8728,E2 307.5823} C_DIS
LIN {X -87.8227,Y 70.2144,Z 116,A 136.1908,B 24.9387,C -1.8084,E1 24.8765,E2 309.7268} C_DIS
LIN {X -85.6847,Y 72.8055,Z 116,A 135.0064,B 24.937,C -1.8334,E1 24.8786,E2 310.8571} C_DIS
LIN {X -83.581,Y 75.2116,Z 116,A 133.1992,B 24.9372,C -1.8306,E1 24.8819,E2 312.6791} C_DIS
LIN {X -80.0056,Y 79.0037,Z 116,A 130.2667,B 24.9375,C -1.8264,E1 24.8877,E2 315.6342} C_DIS
LIN {X -76.3735,Y 82.5216,Z 116,A 127.8753,B 24.9366,C -1.8397,E1 24.8925,E2 318.0038} C_DIS
LIN {X -73.2633,Y 85.2947,Z 116,A 125.5671,B 24.9367,C -1.8373,E1 24.8974,E2 320.3267} C_DIS
LIN {X -68.2166,Y 89.3826,Z 116,A 122.6274,B 24.9352,C -1.8591,E1 24.9037,E2 323.2255} C_DIS
LIN {X -66.2015,Y 90.8841,Z 116,A 121.1525,B 24.9356,C -1.854,E1 24.907,E2 324.7176} C_DIS
LIN {X -61.8848,Y 93.8762,Z 116,A 118.4976,B 24.9351,C -1.8602,E1 24.9132,E2 327.3667} C_DIS
LIN {X -59.0463,Y 95.6891,Z 116,A 116.9146,B 24.9345,C -1.8687,E1 24.9169,E2 328.9344} C_DIS
LIN {X -56.4797,Y 97.2256,Z 116,A 114.2226,B 24.9375,C -1.8254,E1 24.9237,E2 331.7375} C_DIS
LIN {X -50.9699,Y 100.2228,Z 116,A 112.091,B 24.9343,C -1.8728,E1 24.9287,E2 333.7622} C_DIS
LIN {X -47.6593,Y 101.8387,Z 116,A 110.2067,B 24.9341,C -1.8755,E1 24.9334,E2 335.645} C_DIS
LIN {X -40.6203,Y 104.8463,Z 116,A 106.3837,B 24.9334,C -1.8842,E1 24.9432,E2 339.4561} C_DIS
LIN {X -38.2253,Y 105.7422,Z 116,A 104.9339,B 24.9337,C -1.88,E1 24.9471,E2 340.9189} C_DIS
LIN {X -31.3219,Y 107.9902,Z 116,A 101.0295,B 24.934,C -1.8759,E1 24.9575,E2 344.8396} C_DIS
LIN {X -27.5634,Y 109.0089,Z 116,A 99.351,B 24.933,C -1.8904,E1 24.9619,E2 346.4864} C_DIS
LIN {X -24.3609,Y 109.7688,Z 116,A 97.4898,B 24.9334,C -1.8844,E1 24.9671,E2 348.3641} C_DIS
LIN {X -20.4881,Y 110.558,Z 116,A 95.4704,B 24.9334,C -1.8858,E1 24.9726,E2 350.3825} C_DIS
LIN {X -17.1626,Y 111.1212,Z 116,A 93.9406,B 24.9327,C -1.8948,E1 24.9767,E2 351.8923} C_DIS
LIN {X -11.365,Y 111.8635,Z 116,A 90.5963,B 24.9336,C -1.8815,E1 24.9861,E2 355.2705} C_DIS
LIN {X -7.257,Y 112.2048,Z 116,A 88.771,B 24.9328,C -1.8937,E1 24.9911,E2 357.0675} C_DIS
LIN {X -0.9657,Y 112.435,Z 116,A 85.7171,B 24.9323,C -1.901,E1 24.9996,E2 360.1044} C_DIS
LIN {X 3.954,Y 112.3704,Z 116,A 83.0401,B 24.9327,C -1.8943,E1 25.0071,E2 362.7971} C_DIS
LIN {X 10.5395,Y 111.9439,Z 116,A 79.7654,B 24.9325,C -1.8978,E1 25.0162,E2 366.0618} C_DIS
LIN {X 15.0573,Y 111.4277,Z 116,A 77.4384,B 24.9325,C -1.8969,E1 25.0227,E2 368.3892} C_DIS
LIN {X 17.8622,Y 111.0131,Z 116,A 76.0144,B 24.9325,C -1.8974,E1 25.0266,E2 369.8108} C_DIS
LIN {X 20.5417,Y 110.5484,Z 116,A 74.4086,B 24.9332,C -1.8876,E1 25.0311,E2 371.4381} C_DIS
LIN {X 24.6804,Y 109.6986,Z 116,A 72.5003,B 24.9325,C -1.8968,E1 25.0362,E2 373.3219} C_DIS
LIN {X 27.3502,Y 109.0637,Z 116,A 70.898,B 24.9332,C -1.8874,E1 25.0406,E2 374.9443} C_DIS
LIN {X 32.8306,Y 107.5401,Z 116,A 68.2802,B 24.9325,C -1.8973,E1 25.0476,E2 377.5342} C_DIS
LIN {X 36.9894,Y 106.1806,Z 116,A 65.8186,B 24.9334,C -1.8855,E1 25.0541,E2 380.0189} C_DIS
LIN {X 40.8565,Y 104.7535,Z 116,A 64.0325,B 24.9325,C -1.897,E1 25.0587,E2 381.7741} C_DIS
LIN {X 43.301,Y 103.7673,Z 116,A 62.4297,B 24.9334,C -1.8844,E1 25.0629,E2 383.403} C_DIS
LIN {X 46.3919,Y 102.4223,Z 116,A 60.0833,B 24.9355,C -1.8555,E1 25.0691,E2 385.8118} C_DIS
LIN {X 50.5622,Y 100.4311,Z 116,A 58.4676,B 24.9334,C -1.8843,E1 25.0729,E2 387.3553} C_DIS
LIN {X 54.7469,Y 98.2103,Z 116,A 56.1412,B 24.9334,C -1.8848,E1 25.0786,E2 389.6737} C_DIS
LIN {X 57.8881,Y 96.394,Z 116,A 54.2576,B 24.9337,C -1.8806,E1 25.0832,E2 391.5617} C_DIS
LIN {X 60.357,Y 94.8668,Z 116,A 52.6686,B 24.9342,C -1.8735,E1 25.087,E2 393.1623} C_DIS
LIN {X 65.3277,Y 91.5138,Z 116,A 50.0248,B 24.9333,C -1.8864,E1 25.093,E2 395.7665} C_DIS
LIN {X 67.0754,Y 90.2425,Z 116,A 48.4588,B 24.9349,C -1.8641,E1 25.0966,E2 397.3799} C_DIS
LIN {X 69.7869,Y 88.1606,Z 116,A 46.781,B 24.9349,C -1.8637,E1 25.1003,E2 399.0524} C_DIS
LIN {X 72.7451,Y 85.7362,Z 116,A 44.8658,B 24.935,C -1.8614,E1 25.1044,E2 400.9656} C_DIS
LIN {X 78.9252,Y 80.0832,Z 116,A 40.9296,B 24.9346,C -1.8673,E1 25.1125,E2 404.8719} C_DIS
LIN {X 82.9919,Y 75.8609,Z 116,A 37.8028,B 24.9355,C -1.8545,E1 25.1185,E2 408.0154} C_DIS
LIN {X 84.6718,Y 73.9809,Z 116,A 36.3753,B 24.9362,C -1.8452,E1 25.1212,E2 409.4586} C_DIS
LIN {X 86.7851,Y 71.4916,Z 116,A 34.0951,B 24.9383,C -1.814,E1 25.1254,E2 411.8019} C_DIS
LIN {X 89.4741,Y 68.0978,Z 116,A 32.5726,B 24.9366,C -1.8388,E1 25.1278,E2 413.2585} C_DIS
LIN {X 91.2204,Y 65.7389,Z 116,A 30.9794,B 24.9372,C -1.8308,E1 25.1305,E2 414.8631} C_DIS
LIN {X 93.1656,Y 62.9498,Z 116,A 29.4109,B 24.937,C -1.8337,E1 25.1329,E2 416.4169} C_DIS
LIN {X 94.8464,Y 60.3888,Z 116,A 27.5506,B 24.9382,C -1.8162,E1 25.1358,E2 418.3093} C_DIS
LIN {X 97.495,Y 56.0109,Z 116,A 25.0944,B 24.9382,C -1.816,E1 25.1393,E2 420.7533} C_DIS
LIN {X 99.4187,Y 52.5208,Z 116,A 23.1328,B 24.9384,C -1.8135,E1 25.1419,E2 422.7106} C_DIS
LIN {X 101.0459,Y 49.3222,Z 116,A 21.2187,B 24.939,C -1.8044,E1 25.1443,E2 424.6358} C_DIS
LIN {X 102.5158,Y 46.1844,Z 116,A 19.5599,B 24.939,C -1.8042,E1 25.1462,E2 426.2861} C_DIS
LIN {X 104.6769,Y 41.0516,Z 116,A 17.1172,B 24.9383,C -1.8138,E1 25.1488,E2 428.6927} C_DIS
LIN {X 106.3252,Y 36.5776,Z 116,A 14.3872,B 24.9398,C -1.7928,E1 25.1515,E2 431.4568} C_DIS
LIN {X 107.2405,Y 33.7968,Z 116,A 12.6435,B 24.9408,C -1.7769,E1 25.1529,E2 433.2283} C_DIS
LIN {X 108.342,Y 30.0809,Z 116,A 10.9415,B 24.9404,C -1.7832,E1 25.1542,E2 434.9056} C_DIS
LIN {X 109.0626,Y 27.3545,Z 116,A 9.3167,B 24.9413,C -1.7703,E1 25.1554,E2 436.5517} C_DIS
LIN {X 109.9052,Y 23.7358,Z 116,A 7.6737,B 24.9409,C -1.7757,E1 25.1564,E2 438.1722} C_DIS
LIN {X 110.4453,Y 21.0797,Z 116,A 6.2182,B 24.9414,C -1.768,E1 25.1572,E2 439.6374} C_DIS
LIN {X 111.0298,Y 17.7542,Z 116,A 4.0013,B 24.9433,C -1.74,E1 25.1582,E2 441.9073} C_DIS
LIN {X 111.557,Y 14.0597,Z 116,A 2.8192,B 24.9415,C -1.7666,E1 25.1586,E2 443.0197} C_DIS
LIN {X 112.1682,Y 7.7997,Z 116,A -0.3006,B 24.9419,C -1.7602,E1 25.1594,E2 446.1363} C_DIS
LIN {X 112.4192,Y 2.1008,Z 116,A -4.0853,B 24.9452,C -1.7108,E1 25.1598,E2 450.0148} C_DIS
LIN {X 112.4166,Y -2.2425,Z 116,A -5.724,B 24.9439,C -1.7296,E1 25.1598,E2 451.5993} C_DIS
LIN {X 112.091,Y -8.8373,Z 116,A -9.3081,B 24.9453,C -1.7087,E1 25.1591,E2 455.2115} C_DIS
LIN {X 111.7599,Y -12.3547,Z 116,A -10.8577,B 24.9449,C -1.7142,E1 25.1587,E2 456.7391} C_DIS
LIN {X 111.3026,Y -15.9448,Z 116,A -12.6164,B 24.9451,C -1.7121,E1 25.158,E2 458.4923} C_DIS
LIN {X 110.4106,Y -21.2598,Z 116,A -14.977,B 24.9445,C -1.7209,E1 25.1569,E2 460.8183} C_DIS
LIN {X 109.7079,Y -24.6402,Z 116,A -17.1536,B 24.9461,C -1.696,E1 25.1556,E2 463.0409} C_DIS
LIN {X 108.9585,Y -27.7593,Z 116,A -18.6878,B 24.9461,C -1.6954,E1 25.1546,E2 464.5676} C_DIS
LIN {X 107.7374,Y -32.1741,Z 116,A -21.1177,B 24.9469,C -1.6836,E1 25.1527,E2 467.0115} C_DIS
LIN {X 106.5076,Y -36.0366,Z 116,A -23.1088,B 24.9471,C -1.6804,E1 25.151,E2 468.9988} C_DIS
LIN {X 105.1879,Y -39.7241,Z 116,A -25.0805,B 24.9474,C -1.6753,E1 25.1491,E2 470.9715} C_DIS
LIN {X 104.0161,Y -42.6995,Z 116,A -26.7294,B 24.9478,C -1.6693,E1 25.1474,E2 472.6254} C_DIS
LIN {X 102.546,Y -46.1173,Z 116,A -29.1946,B 24.9497,C -1.6377,E1 25.1445,E2 475.1517} C_DIS
LIN {X 100.6954,Y -50.0292,Z 116,A -30.5186,B 24.9477,C -1.6711,E1 25.143,E2 476.3901} C_DIS
LIN {X 99.6596,Y -52.0628,Z 116,A -32.3525,B 24.9498,C -1.6371,E1 25.1406,E2 478.2943} C_DIS
LIN {X 97.9789,Y -55.1613,Z 116,A -33.6404,B 24.9487,C -1.6548,E1 25.1389,E2 479.5337} C_DIS
LIN {X 96.3835,Y -57.9053,Z 116,A -36.0404,B 24.9511,C -1.6147,E1 25.1353,E2 482.016} C_DIS
LIN {X 93.8652,Y -61.9016,Z 116,A -37.3254,B 24.9484,C -1.6586,E1 25.1336,E2 483.191} C_DIS
LIN {X 92.3789,Y -64.0985,Z 116,A -39.0795,B 24.9498,C -1.6365,E1 25.1307,E2 484.9887} C_DIS
LIN {X 90.2932,Y -67.0079,Z 116,A -40.9286,B 24.9502,C -1.6303,E1 25.1277,E2 486.8435} C_DIS
LIN {X 88.1492,Y -69.8013,Z 116,A -42.6348,B 24.9502,C -1.6294,E1 25.1247,E2 488.5436} C_DIS
LIN {X 86.0399,Y -72.3884,Z 116,A -44.488,B 24.9509,C -1.618,E1 25.1214,E2 490.4152} C_DIS
LIN {X 83.5664,Y -75.2279,Z 116,A -46.2452,B 24.9509,C -1.6204,E1 25.1182,E2 492.159} C_DIS
LIN {X 81.1585,Y -77.8195,Z 116,A -48.0722,B 24.9511,C -1.6147,E1 25.1147,E2 493.9913} C_DIS
LIN {X 78.7673,Y -80.2392,Z 116,A -49.7324,B 24.9512,C -1.6138,E1 25.1114,E2 495.6468} C_DIS
LIN {X 76.2399,Y -82.6441,Z 116,A -51.5606,B 24.9516,C -1.6073,E1 25.1077,E2 497.4829} C_DIS
LIN {X 73.9298,Y -84.7164,Z 116,A -52.9412,B 24.9513,C -1.6126,E1 25.1048,E2 498.8453} C_DIS
LIN {X 71.8485,Y -86.4886,Z 116,A -54.4892,B 24.9519,C -1.6025,E1 25.1015,E2 500.4113} C_DIS
LIN {X 69.2657,Y -88.5724,Z 116,A -56.2177,B 24.9522,C -1.5971,E1 25.0977,E2 502.1461} C_DIS
LIN {X 66.4777,Y -90.6819,Z 116,A -57.9466,B 24.9522,C -1.5956,E1 25.0938,E2 503.8722} C_DIS
LIN {X 63.7224,Y -92.6404,Z 116,A -59.6291,B 24.9524,C -1.5939,E1 25.09,E2 505.5531} C_DIS
LIN {X 57.8331,Y -96.4272,Z 116,A -63.1477,B 24.9527,C -1.5891,E1 25.0817,E2 509.0716} C_DIS
LIN {X 55.501,Y -97.7879,Z 116,A -64.5842,B 24.953,C -1.5839,E1 25.0782,E2 510.516} C_DIS
LIN {X 52.6119,Y -99.3707,Z 116,A -66.3564,B 24.9534,C -1.5769,E1 25.0738,E2 512.2998} C_DIS
LIN {X 48.0857,Y -101.6401,Z 116,A -68.8708,B 24.9534,C -1.5755,E1 25.0675,E2 514.8108} C_DIS
LIN {X 45.0427,Y -103.0226,Z 116,A -70.5379,B 24.9536,C -1.5745,E1 25.0632,E2 516.4761} C_DIS
LIN {X 42.0991,Y -104.2605,Z 116,A -73.1225,B 24.9561,C -1.5305,E1 25.0563,E2 519.159} C_DIS
LIN {X 36.5728,Y -106.3268,Z 116,A -75.0883,B 24.9537,C -1.5717,E1 25.0514,E2 521.0233} C_DIS
LIN {X 33.0397,Y -107.4753,Z 116,A -77.1441,B 24.9543,C -1.5623,E1 25.0459,E2 523.0975} C_DIS
LIN {X 29.3864,Y -108.5308,Z 116,A -78.9882,B 24.9542,C -1.5643,E1 25.0409,E2 524.9339} C_DIS
LIN {X 26.0945,Y -109.3704,Z 116,A -80.6442,B 24.9541,C -1.5658,E1 25.0365,E2 526.5839} C_DIS
LIN {X 21.3995,Y -110.3837,Z 116,A -82.8302,B 24.9535,C -1.575,E1 25.0306,E2 528.7454} C_DIS
LIN {X 16.5798,Y -111.2113,Z 116,A -85.5705,B 24.9543,C -1.5622,E1 25.023,E2 531.5131} C_DIS
LIN {X 13.4769,Y -111.6289,Z 116,A -87.8663,B 24.9561,C -1.5312,E1 25.0164,E2 533.8805} C_DIS
LIN {X 9.1143,Y -112.0689,Z 116,A -89.2887,B 24.9541,C -1.5648,E1 25.0127,E2 535.2226} C_DIS
LIN {X 3.0564,Y -112.3979,Z 116,A -92.5655,B 24.9547,C -1.5556,E1 25.0035,E2 538.52} C_DIS
LIN {X 0.8058,Y -112.4294,Z 116,A -94.1431,B 24.9557,C -1.5371,E1 24.9989,E2 540.1414} C_DIS
Enddeposition()
LIN {X 0.8058,Y -112.4294,Z 116,A -94.1431,B 24.9557,C -1.5371,E1 24.9989,E2 540.1414} C_DIS
Startdeposition()
$VEL.CP = VEL_PRINT
LIN {X 2.4531,Y -111.5054,Z 116,A -92.1369,B 24.9519,C -1.6026,E1 25.005,E2 537.9802} C_DIS
LIN {X 5.7953,Y -111.3816,Z 116,A -90.3343,B 24.9516,C -1.6068,E1 25.01,E2 536.168} C_DIS
LIN {X 10.0974,Y -111.0737,Z 116,A -87.8397,B 24.9508,C -1.62,E1 25.017,E2 533.6434} C_DIS
LIN {X 15.1952,Y -110.4928,Z 116,A -85.3981,B 24.9512,C -1.6132,E1 25.0237,E2 531.2199} C_DIS
LIN {X 18.1345,Y -110.0478,Z 116,A -83.6862,B 24.9507,C -1.6225,E1 25.0285,E2 529.4878} C_DIS
LIN {X 21.8365,Y -109.3748,Z 116,A -81.8209,B 24.9507,C -1.6211,E1 25.0336,E2 527.628} C_DIS
LIN {X 26.2749,Y -108.3926,Z 116,A -79.751,B 24.9513,C -1.6118,E1 25.0392,E2 525.5831} C_DIS
LIN {X 29.7524,Y -107.4916,Z 116,A -77.8767,B 24.9511,C -1.615,E1 25.0442,E2 523.7042} C_DIS
LIN {X 32.767,Y -106.6101,Z 116,A -76.3122,B 24.9511,C -1.6147,E1 25.0484,E2 522.1431} C_DIS
LIN {X 36.2592,Y -105.4752,Z 116,A -73.868,B 24.9495,C -1.6417,E1 25.055,E2 519.6397} C_DIS
LIN {X 40.0796,Y -104.0832,Z 116,A -72.3946,B 24.951,C -1.6173,E1 25.0587,E2 518.2273} C_DIS
LIN {X 42.933,Y -102.938,Z 116,A -70.7557,B 24.9507,C -1.6222,E1 25.063,E2 516.5806} C_DIS
LIN {X 45.658,Y -101.758,Z 116,A -69.1987,B 24.9505,C -1.626,E1 25.067,E2 515.0185} C_DIS
LIN {X 48.8816,Y -100.2512,Z 116,A -67.2401,B 24.9499,C -1.6347,E1 25.0719,E2 513.0444} C_DIS
Enddeposition()
END
